KUKA KRL program: MyProgram_131().src

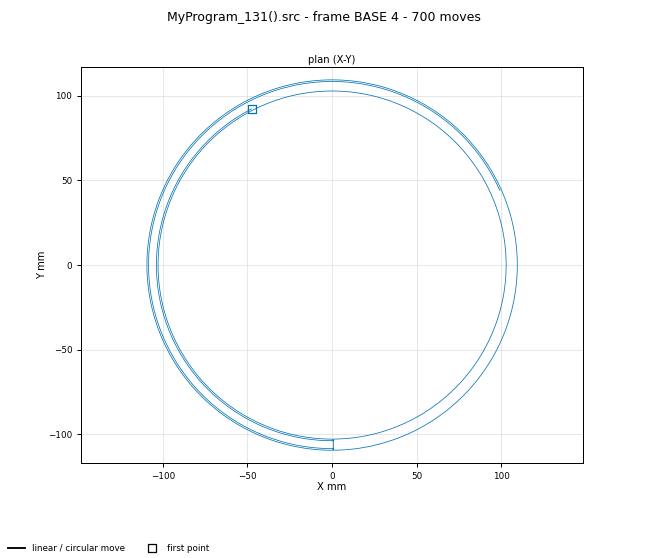
[picture p0: tool path of MyProgram_131().src in frame BASE 4, 700 of 700 moves have a stored position in this frame; points joined in program order, loops and branches not executed]
&ACCESS RVP
&REL 1
&PARAM TEMPLATE = C:\KRC\Roboter\Template\vorgabe
&PARAM EDITMASK = *
DEF MyProgram_131()
; ---- Setting reference (Base) ----
$BASE = BASE_DATA[4]

; --------------------------
; ---- Setting tool (TCP) ----
$TOOL = TOOL_DATA[3]
; --------------------------

$VEL.CP = VEL_APROX_PRINT
Startdeposition()
$VEL.CP = VEL_PRINT
LIN {X -47.5372,Y 92.2572,Z 107,A 112.7806,B 24.923,C -2.027,E1 24.926,E2 332.7039} C_DIS
LIN {X -49.4376,Y 91.2522,Z 107,A 114.1175,B 24.9227,C -2.0305,E1 24.9227,E2 331.3549} C_DIS
LIN {X -54.474,Y 88.3398,Z 107,A 117.7592,B 24.9219,C -2.0405,E1 24.9139,E2 327.6784} C_DIS
LIN {X -57.2487,Y 86.5659,Z 107,A 119.0499,B 24.9237,C -2.0176,E1 24.911,E2 326.4379} C_DIS
LIN {X -60.0172,Y 84.6705,Z 107,A 121.0764,B 24.9235,C -2.0203,E1 24.9063,E2 324.3982} C_DIS
LIN {X -63.2144,Y 82.3105,Z 107,A 123.2686,B 24.9238,C -2.0156,E1 24.9014,E2 322.2093} C_DIS
LIN {X -66.0188,Y 80.0795,Z 107,A 125.2015,B 24.9243,C -2.0096,E1 24.8973,E2 320.2834} C_DIS
LIN {X -68.7354,Y 77.7617,Z 107,A 127.217,B 24.9245,C -2.0067,E1 24.893,E2 318.2668} C_DIS
LIN {X -70.7621,Y 75.9209,Z 107,A 128.5161,B 24.9253,C -1.9956,E1 24.8904,E2 316.9891} C_DIS
LIN {X -72.935,Y 73.8345,Z 107,A 130.3237,B 24.9253,C -1.9968,E1 24.8867,E2 315.171} C_DIS
LIN {X -75.0796,Y 71.6545,Z 107,A 132.1843,B 24.9251,C -1.9988,E1 24.8831,E2 313.2975} C_DIS
LIN {X -77.6382,Y 68.8736,Z 107,A 134.0763,B 24.926,C -1.9866,E1 24.8796,E2 311.4263} C_DIS
LIN {X -79.2084,Y 67.061,Z 107,A 135.593,B 24.9257,C -1.9901,E1 24.8768,E2 309.8943} C_DIS
LIN {X -81.5466,Y 64.1968,Z 107,A 137.5851,B 24.9263,C -1.9829,E1 24.8734,E2 307.91} C_DIS
LIN {X -83.4567,Y 61.6949,Z 107,A 139.3497,B 24.9266,C -1.9792,E1 24.8704,E2 306.1458} C_DIS
LIN {X -85.5785,Y 58.7177,Z 107,A 141.2336,B 24.9273,C -1.9688,E1 24.8674,E2 304.2774} C_DIS
LIN {X -87.4411,Y 55.903,Z 107,A 143.96,B 24.9254,C -1.9945,E1 24.8632,E2 301.4758} C_DIS
LIN {X -89.8473,Y 51.948,Z 107,A 145.8018,B 24.9279,C -1.9615,E1 24.8607,E2 299.7033} C_DIS
LIN {X -91.4843,Y 49.0098,Z 107,A 148.2104,B 24.9268,C -1.9758,E1 24.8574,E2 297.2478} C_DIS
LIN {X -93.2578,Y 45.5457,Z 107,A 149.9432,B 24.9284,C -1.9545,E1 24.8554,E2 295.5565} C_DIS
LIN {X -94.9695,Y 41.8571,Z 107,A 151.8784,B 24.9297,C -1.9367,E1 24.8531,E2 293.6531} C_DIS
LIN {X -96.1628,Y 39.0355,Z 107,A 153.7151,B 24.9297,C -1.9367,E1 24.8512,E2 291.8063} C_DIS
LIN {X -97.0153,Y 36.8659,Z 107,A 155.0952,B 24.9297,C -1.936,E1 24.8498,E2 290.42} C_DIS
LIN {X -98.5087,Y 32.6703,Z 107,A 157.459,B 24.9305,C -1.925,E1 24.8476,E2 288.0691} C_DIS
LIN {X -99.5427,Y 29.3653,Z 107,A 159.4752,B 24.9307,C -1.9227,E1 24.846,E2 286.0467} C_DIS
LIN {X -100.6094,Y 25.4744,Z 107,A 161.5957,B 24.9315,C -1.9118,E1 24.8445,E2 283.9398} C_DIS
LIN {X -101.6647,Y 20.8647,Z 107,A 164.1136,B 24.9323,C -1.9002,E1 24.843,E2 281.4348} C_DIS
LIN {X -102.1521,Y 18.3302,Z 107,A 165.7626,B 24.9321,C -1.9035,E1 24.8421,E2 279.7681} C_DIS
LIN {X -102.734,Y 14.7241,Z 107,A 167.7191,B 24.9327,C -1.8949,E1 24.8413,E2 277.8206} C_DIS
LIN {X -103.1383,Y 11.5673,Z 107,A 169.4687,B 24.9331,C -1.889,E1 24.8407,E2 276.0746} C_DIS
LIN {X -103.3969,Y 8.9692,Z 107,A 171.1174,B 24.9329,C -1.8916,E1 24.8403,E2 274.4097} C_DIS
LIN {X -103.663,Y 5.0357,Z 107,A 173.3276,B 24.9333,C -1.8858,E1 24.8399,E2 272.2002} C_DIS
LIN {X -103.7792,Y 1.0625,Z 107,A 175.5136,B 24.9339,C -1.8784,E1 24.8398,E2 270.0186} C_DIS
LIN {X -103.7423,Y -2.9396,Z 107,A 177.7377,B 24.9343,C -1.8718,E1 24.8399,E2 267.7969} C_DIS
LIN {X -103.598,Y -6.2259,Z 107,A 179.5759,B 24.9347,C -1.8667,E1 24.8402,E2 265.9596} C_DIS
LIN {X -103.343,Y -9.5537,Z 107,A -178.6602,B 24.9353,C -1.8581,E1 24.8406,E2 264.2059} C_DIS
LIN {X -103.0312,Y -12.4821,Z 107,A -176.9436,B 24.9354,C -1.8561,E1 24.8412,E2 262.4836} C_DIS
LIN {X -102.5449,Y -15.9876,Z 107,A -175.0994,B 24.9361,C -1.8461,E1 24.8419,E2 260.6525} C_DIS
LIN {X -101.9172,Y -19.5943,Z 107,A -173.0077,B 24.9364,C -1.8422,E1 24.8429,E2 258.5575} C_DIS
LIN {X -101.3208,Y -22.4785,Z 107,A -171.4793,B 24.937,C -1.8337,E1 24.8438,E2 257.0404} C_DIS
LIN {X -100.5441,Y -25.7282,Z 107,A -169.5554,B 24.9372,C -1.8308,E1 24.8451,E2 255.1121} C_DIS
LIN {X -99.4164,Y -29.7911,Z 107,A -167.0771,B 24.9372,C -1.8291,E1 24.847,E2 252.6236} C_DIS
LIN {X -98.176,Y -33.6571,Z 107,A -164.8048,B 24.9377,C -1.8235,E1 24.849,E2 250.3518} C_DIS
LIN {X -96.8184,Y -37.3847,Z 107,A -162.589,B 24.9381,C -1.8179,E1 24.8512,E2 248.1366} C_DIS
LIN {X -95.3011,Y -41.0964,Z 107,A -160.5252,B 24.9389,C -1.8062,E1 24.8534,E2 246.0895} C_DIS
LIN {X -94.0744,Y -43.83,Z 107,A -158.8309,B 24.9391,C -1.8029,E1 24.8554,E2 244.3936} C_DIS
LIN {X -92.7841,Y -46.5012,Z 107,A -157.1505,B 24.9393,C -1.7999,E1 24.8575,E2 242.7115} C_DIS
LIN {X -90.1144,Y -51.4831,Z 107,A -154.2992,B 24.9405,C -1.7816,E1 24.8613,E2 239.8886} C_DIS
LIN {X -88.6267,Y -54.0034,Z 107,A -152.3658,B 24.94,C -1.7888,E1 24.8641,E2 237.9281} C_DIS
LIN {X -86.5659,Y -57.2487,Z 107,A -150.3857,B 24.9407,C -1.7781,E1 24.867,E2 235.9634} C_DIS
LIN {X -84.9538,Y -59.6164,Z 107,A -148.7985,B 24.941,C -1.7743,E1 24.8696,E2 234.3775} C_DIS
LIN {X -83.2306,Y -61.9991,Z 107,A -147.2699,B 24.9415,C -1.7669,E1 24.8721,E2 232.8592} C_DIS
LIN {X -81.4412,Y -64.3303,Z 107,A -145.4019,B 24.9412,C -1.7719,E1 24.8753,E2 230.9704} C_DIS
LIN {X -78.951,Y -67.3631,Z 107,A -143.2259,B 24.9415,C -1.7672,E1 24.8792,E2 228.7956} C_DIS
LIN {X -75.7408,Y -70.9536,Z 107,A -140.5603,B 24.9418,C -1.7615,E1 24.8842,E2 226.1318} C_DIS
LIN {X -73.0815,Y -73.6898,Z 107,A -138.0497,B 24.9412,C -1.7719,E1 24.8892,E2 223.5857} C_DIS
LIN {X -70.6358,Y -76.0396,Z 107,A -136.6878,B 24.9427,C -1.7492,E1 24.8919,E2 222.2724} C_DIS
LIN {X -68.8518,Y -77.6578,Z 107,A -135.1448,B 24.9423,C -1.7544,E1 24.8952,E2 220.7107} C_DIS
LIN {X -65.9356,Y -80.1487,Z 107,A -133.0147,B 24.9425,C -1.7509,E1 24.8997,E2 218.5809} C_DIS
LIN {X -63.4404,Y -82.1364,Z 107,A -131.372,B 24.943,C -1.7433,E1 24.9033,E2 216.9502} C_DIS
LIN {X -61.1951,Y -83.8226,Z 107,A -129.7963,B 24.9432,C -1.7416,E1 24.9068,E2 215.3731} C_DIS
LIN {X -58.2223,Y -85.914,Z 107,A -127.7657,B 24.9433,C -1.7391,E1 24.9115,E2 213.3413} C_DIS
LIN {X -55.7846,Y -87.5171,Z 107,A -126.1028,B 24.9433,C -1.7386,E1 24.9154,E2 211.6744} C_DIS
LIN {X -53.0914,Y -89.1766,Z 107,A -124.4049,B 24.9436,C -1.7342,E1 24.9195,E2 209.9818} C_DIS
LIN {X -49.2389,Y -91.36,Z 107,A -122.0744,B 24.9441,C -1.7265,E1 24.9251,E2 207.6627} C_DIS
LIN {X -46.3808,Y -92.8438,Z 107,A -120.1017,B 24.9438,C -1.7316,E1 24.9301,E2 205.6725} C_DIS
LIN {X -43.7788,Y -94.0982,Z 107,A -118.5776,B 24.9441,C -1.7271,E1 24.9339,E2 204.1554} C_DIS
LIN {X -40.3364,Y -95.6244,Z 107,A -116.4884,B 24.9442,C -1.7253,E1 24.9393,E2 202.0656} C_DIS
LIN {X -36.9737,Y -96.9745,Z 107,A -113.8939,B 24.9429,C -1.7461,E1 24.9462,E2 199.416} C_DIS
LIN {X -33.1975,Y -98.3309,Z 107,A -112.3467,B 24.9446,C -1.7186,E1 24.9501,E2 197.9313} C_DIS
LIN {X -30.1841,Y -99.299,Z 107,A -110.4082,B 24.9443,C -1.7246,E1 24.9553,E2 195.9751} C_DIS
LIN {X -26.4931,Y -100.347,Z 107,A -108.4997,B 24.9449,C -1.7152,E1 24.9604,E2 194.0861} C_DIS
LIN {X -23.4588,Y -101.0977,Z 107,A -106.603,B 24.9445,C -1.7209,E1 24.9656,E2 192.1732} C_DIS
LIN {X -19.4848,Y -101.9383,Z 107,A -104.3957,B 24.9446,C -1.7186,E1 24.9716,E2 189.9688} C_DIS
LIN {X -16.5691,Y -102.454,Z 107,A -102.6676,B 24.9444,C -1.7217,E1 24.9764,E2 188.2317} C_DIS
LIN {X -12.6661,Y -103.0096,Z 107,A -100.4703,B 24.9444,C -1.7221,E1 24.9825,E2 186.0318} C_DIS
LIN {X -8.6432,Y -103.4238,Z 107,A -98.2815,B 24.9445,C -1.7203,E1 24.9886,E2 183.8463} C_DIS
LIN {X -5.0186,Y -103.6638,Z 107,A -96.2028,B 24.9443,C -1.7232,E1 24.9944,E2 181.76} C_DIS
LIN {X -1.2387,Y -103.778,Z 107,A -94.3648,B 24.945,C -1.7137,E1 24.9995,E2 179.9443} C_DIS
LIN {X 0.7183,Y -103.7767,Z 107,A -93.2927,B 24.945,C -1.7137,E1 25.0025,E2 178.8722} C_DIS
Enddeposition()
LIN {X 0.7183,Y -103.7767,Z 107,A -93.2927,B 24.945,C -1.7137,E1 25.0025,E2 178.8722} C_DIS
Startdeposition()
$VEL.CP = VEL_PRINT
LIN {X -0.0761,Y -102.8201,Z 107,A -94.3958,B 24.9455,C -1.7047,E1 24.9993,E2 179.9968} C_DIS
LIN {X -2.5322,Y -102.7893,Z 107,A -95.9772,B 24.9461,C -1.6963,E1 24.9948,E2 181.5982} C_DIS
LIN {X -6.5744,Y -102.6089,Z 107,A -97.9527,B 24.9454,C -1.7068,E1 24.9894,E2 183.5492} C_DIS
LIN {X -8.8274,Y -102.4409,Z 107,A -99.4199,B 24.9459,C -1.6989,E1 24.9853,E2 185.0359} C_DIS
LIN {X -11.4014,Y -102.1861,Z 107,A -100.9306,B 24.9461,C -1.6964,E1 24.9811,E2 186.5534} C_DIS
LIN {X -15.1469,Y -101.6984,Z 107,A -102.8262,B 24.9455,C -1.7048,E1 24.9759,E2 188.4305} C_DIS
LIN {X -17.6331,Y -101.297,Z 107,A -104.2774,B 24.9456,C -1.7034,E1 24.9718,E2 189.8864} C_DIS
LIN {X -20.1263,Y -100.8311,Z 107,A -105.6747,B 24.9456,C -1.7046,E1 24.968,E2 191.2825} C_DIS
LIN {X -22.981,Y -100.2176,Z 107,A -107.1134,B 24.945,C -1.7125,E1 24.9641,E2 192.7043} C_DIS
LIN {X -25.0414,Y -99.7242,Z 107,A -108.4562,B 24.9454,C -1.707,E1 24.9605,E2 194.062} C_DIS
LIN {X -27.4771,Y -99.0808,Z 107,A -109.8639,B 24.9454,C -1.7077,E1 24.9567,E2 195.4701} C_DIS
LIN {X -30.3817,Y -98.2274,Z 107,A -111.6646,B 24.9455,C -1.7047,E1 24.9518,E2 197.2811} C_DIS
LIN {X -33.4794,Y -97.2171,Z 107,A -113.4221,B 24.9453,C -1.7083,E1 24.9472,E2 199.0332} C_DIS
LIN {X -35.8853,Y -96.3548,Z 107,A -114.8015,B 24.9451,C -1.7112,E1 24.9436,E2 200.4084} C_DIS
LIN {X -38.2411,Y -95.4443,Z 107,A -116.2076,B 24.9451,C -1.7126,E1 24.9399,E2 201.8143} C_DIS
LIN {X -40.566,Y -94.4796,Z 107,A -117.6131,B 24.9449,C -1.714,E1 24.9363,E2 203.2197} C_DIS
LIN {X -42.8147,Y -93.4824,Z 107,A -119.0182,B 24.9449,C -1.7142,E1 24.9327,E2 204.6277} C_DIS
LIN {X -45.158,Y -92.3729,Z 107,A -120.4656,B 24.9449,C -1.7159,E1 24.9291,E2 206.0749} C_DIS
LIN {X -47.3577,Y -91.265,Z 107,A -121.9236,B 24.9449,C -1.7144,E1 24.9254,E2 207.5402} C_DIS
LIN {X -49.6955,Y -90.0126,Z 107,A -123.2777,B 24.9445,C -1.721,E1 24.9221,E2 208.8826} C_DIS
LIN {X -51.8837,Y -88.7694,Z 107,A -124.6718,B 24.9443,C -1.7233,E1 24.9188,E2 210.2754} C_DIS
LIN {X -53.9437,Y -87.5337,Z 107,A -126.2088,B 24.9447,C -1.718,E1 24.9151,E2 211.8297} C_DIS
LIN {X -56.1184,Y -86.1552,Z 107,A -127.4851,B 24.9442,C -1.726,E1 24.9121,E2 213.0911} C_DIS
LIN {X -58.2109,Y -84.7555,Z 107,A -128.8962,B 24.944,C -1.728,E1 24.9088,E2 214.5022} C_DIS
LIN {X -60.2359,Y -83.3289,Z 107,A -130.3077,B 24.944,C -1.7292,E1 24.9056,E2 215.9157} C_DIS
LIN {X -62.724,Y -81.4701,Z 107,A -132.0601,B 24.9438,C -1.7315,E1 24.9017,E2 217.669} C_DIS
LIN {X -64.7681,Y -79.8546,Z 107,A -133.6037,B 24.9438,C -1.7308,E1 24.8983,E2 219.2199} C_DIS
LIN {X -67.1843,Y -77.835,Z 107,A -135.3788,B 24.9437,C -1.7334,E1 24.8946,E2 220.9956} C_DIS
LIN {X -69.5343,Y -75.7407,Z 107,A -137.0324,B 24.9432,C -1.7406,E1 24.8911,E2 222.6389} C_DIS
LIN {X -71.8178,Y -73.5816,Z 107,A -138.9911,B 24.9435,C -1.7368,E1 24.8872,E2 224.6148} C_DIS
LIN {X -74.1781,Y -71.1992,Z 107,A -140.7928,B 24.943,C -1.7432,E1 24.8837,E2 226.4089} C_DIS
LIN {X -76.611,Y -68.5743,Z 107,A -142.6677,B 24.9425,C -1.7519,E1 24.8802,E2 228.2713} C_DIS
LIN {X -78.2864,Y -66.6551,Z 107,A -144.1941,B 24.9425,C -1.7514,E1 24.8774,E2 229.8059} C_DIS
LIN {X -80.2918,Y -64.2283,Z 107,A -146.0563,B 24.9425,C -1.7517,E1 24.8741,E2 231.676} C_DIS
LIN {X -82.6132,Y -61.2134,Z 107,A -147.997,B 24.9417,C -1.7632,E1 24.8708,E2 233.5986} C_DIS
LIN {X -84.0655,Y -59.2035,Z 107,A -149.5834,B 24.942,C -1.7594,E1 24.8682,E2 235.2017} C_DIS
LIN {X -85.9185,Y -56.4775,Z 107,A -151.3261,B 24.9414,C -1.7675,E1 24.8656,E2 236.9339} C_DIS
LIN {X -87.5689,Y -53.8857,Z 107,A -152.9474,B 24.9409,C -1.7752,E1 24.8632,E2 238.5452} C_DIS
LIN {X -88.8623,Y -51.7252,Z 107,A -154.3501,B 24.9407,C -1.7789,E1 24.8612,E2 239.9462} C_DIS
LIN {X -90.0887,Y -49.5588,Z 107,A -155.7774,B 24.9405,C -1.7813,E1 24.8592,E2 241.3754} C_DIS
LIN {X -91.2661,Y -47.3557,Z 107,A -157.1569,B 24.9402,C -1.7855,E1 24.8574,E2 242.7521} C_DIS
LIN {X -92.4269,Y -45.0474,Z 107,A -158.7861,B 24.9404,C -1.7829,E1 24.8554,E2 244.3963} C_DIS
LIN {X -93.8431,Y -42.0144,Z 107,A -160.5575,B 24.9398,C -1.7915,E1 24.8534,E2 246.1569} C_DIS
LIN {X -94.9956,Y -39.3433,Z 107,A -162.1397,B 24.9394,C -1.7976,E1 24.8516,E2 247.7335} C_DIS
LIN {X -95.9307,Y -37.0049,Z 107,A -163.5255,B 24.9391,C -1.8023,E1 24.8502,E2 249.1158} C_DIS
LIN {X -96.8333,Y -34.573,Z 107,A -164.9482,B 24.9388,C -1.8073,E1 24.8489,E2 250.5345} C_DIS
LIN {X -97.6884,Y -32.0756,Z 107,A -166.3649,B 24.9383,C -1.8136,E1 24.8476,E2 251.9443} C_DIS
LIN {X -98.4067,Y -29.8015,Z 107,A -167.7742,B 24.9383,C -1.8148,E1 24.8464,E2 253.3588} C_DIS
LIN {X -99.1052,Y -27.3894,Z 107,A -169.257,B 24.9382,C -1.8162,E1 24.8453,E2 254.8469} C_DIS
LIN {X -99.7408,Y -24.9767,Z 107,A -170.6348,B 24.9378,C -1.8209,E1 24.8444,E2 256.2215} C_DIS
LIN {X -100.3228,Y -22.5256,Z 107,A -172.0196,B 24.9375,C -1.8259,E1 24.8435,E2 257.6025} C_DIS
LIN {X -100.8554,Y -20.0046,Z 107,A -173.4376,B 24.9372,C -1.831,E1 24.8427,E2 259.0167} C_DIS
LIN {X -101.3154,Y -17.5268,Z 107,A -175.0708,B 24.9374,C -1.8275,E1 24.8419,E2 260.6679} C_DIS
LIN {X -101.8931,Y -13.7765,Z 107,A -176.9788,B 24.9364,C -1.8413,E1 24.8411,E2 262.5544} C_DIS
LIN {X -102.2,Y -11.276,Z 107,A -178.4221,B 24.9362,C -1.8444,E1 24.8407,E2 263.9989} C_DIS
LIN {X -102.441,Y -8.826,Z 107,A -179.8044,B 24.936,C -1.8484,E1 24.8403,E2 265.3799} C_DIS
LIN {X -102.6593,Y -5.722,Z 107,A 178.6127,B 24.9352,C -1.8593,E1 24.84,E2 266.9466} C_DIS
LIN {X -102.7529,Y -3.7192,Z 107,A 177.3254,B 24.9354,C -1.8569,E1 24.8399,E2 268.2471} C_DIS
LIN {X -102.8138,Y -1.1098,Z 107,A 175.9089,B 24.9349,C -1.8629,E1 24.8398,E2 269.6578} C_DIS
LIN {X -102.811,Y 1.3581,Z 107,A 174.524,B 24.9347,C -1.867,E1 24.8398,E2 271.0413} C_DIS
LIN {X -102.7487,Y 3.8348,Z 107,A 173.0516,B 24.9346,C -1.8683,E1 24.8399,E2 272.5195} C_DIS
LIN {X -102.6227,Y 6.3692,Z 107,A 171.6611,B 24.9342,C -1.8737,E1 24.8402,E2 273.9055} C_DIS
LIN {X -102.3252,Y 10.0809,Z 107,A 169.5429,B 24.9338,C -1.8789,E1 24.8407,E2 276.024} C_DIS
LIN {X -102.0475,Y 12.5851,Z 107,A 168.1561,B 24.9335,C -1.8841,E1 24.8411,E2 277.4069} C_DIS
LIN {X -101.6997,Y 15.1383,Z 107,A 166.7368,B 24.9331,C -1.8893,E1 24.8417,E2 278.8222} C_DIS
LIN {X -101.2071,Y 18.133,Z 107,A 164.9234,B 24.933,C -1.8905,E1 24.8425,E2 280.6434} C_DIS
LIN {X -100.5717,Y 21.3843,Z 107,A 163.1798,B 24.9323,C -1.8999,E1 24.8435,E2 282.3748} C_DIS
LIN {X -100.0195,Y 23.8343,Z 107,A 161.7411,B 24.9321,C -1.903,E1 24.8444,E2 283.8146} C_DIS
LIN {X -99.4221,Y 26.2164,Z 107,A 160.3347,B 24.9319,C -1.9061,E1 24.8454,E2 285.2219} C_DIS
LIN {X -98.6158,Y 29.0968,Z 107,A 158.8866,B 24.931,C -1.9189,E1 24.8465,E2 286.6477} C_DIS
LIN {X -98.0043,Y 31.0994,Z 107,A 157.5095,B 24.9312,C -1.9153,E1 24.8476,E2 288.0414} C_DIS
LIN {X -97.2249,Y 33.4571,Z 107,A 156.0898,B 24.931,C -1.9184,E1 24.8489,E2 289.4619} C_DIS
LIN {X -96.3582,Y 35.8761,Z 107,A 154.6667,B 24.9307,C -1.9231,E1 24.8502,E2 290.8817} C_DIS
LIN {X -95.4461,Y 38.2365,Z 107,A 153.2833,B 24.9303,C -1.9284,E1 24.8516,E2 292.2603} C_DIS
LIN {X -94.4808,Y 40.5632,Z 107,A 151.8691,B 24.93,C -1.9323,E1 24.8532,E2 293.673} C_DIS
LIN {X -93.483,Y 42.8135,Z 107,A 150.4306,B 24.9299,C -1.9341,E1 24.8548,E2 295.115} C_DIS
LIN {X -92.3594,Y 45.1851,Z 107,A 148.8658,B 24.9299,C -1.935,E1 24.8567,E2 296.6863} C_DIS
LIN {X -91.2582,Y 47.3707,Z 107,A 147.5902,B 24.9293,C -1.9421,E1 24.8583,E2 297.9518} C_DIS
LIN {X -89.9448,Y 49.817,Z 107,A 145.9803,B 24.9291,C -1.9444,E1 24.8605,E2 299.5646} C_DIS
LIN {X -88.203,Y 52.842,Z 107,A 144.0992,B 24.9285,C -1.9523,E1 24.8631,E2 301.4367} C_DIS
LIN {X -86.866,Y 55.0124,Z 107,A 142.6426,B 24.9283,C -1.955,E1 24.8653,E2 302.8942} C_DIS
LIN {X -85.4922,Y 57.124,Z 107,A 141.2293,B 24.9281,C -1.9586,E1 24.8675,E2 304.306} C_DIS
LIN {X -83.7242,Y 59.6819,Z 107,A 139.4889,B 24.9277,C -1.9632,E1 24.8702,E2 306.0441} C_DIS
LIN {X -81.8245,Y 62.2641,Z 107,A 137.5093,B 24.9279,C -1.9613,E1 24.8736,E2 308.0378} C_DIS
LIN {X -79.8595,Y 64.7621,Z 107,A 135.8362,B 24.9273,C -1.9694,E1 24.8765,E2 309.6993} C_DIS
LIN {X -77.5417,Y 67.5202,Z 107,A 133.8707,B 24.9268,C -1.976,E1 24.88,E2 311.6579} C_DIS
LIN {X -75.7336,Y 69.5421,Z 107,A 132.296,B 24.9267,C -1.9777,E1 24.883,E2 313.2358} C_DIS
LIN {X -73.5691,Y 71.8305,Z 107,A 130.435,B 24.9267,C -1.9782,E1 24.8866,E2 315.1034} C_DIS
LIN {X -71.334,Y 74.0482,Z 107,A 128.7682,B 24.9261,C -1.9856,E1 24.8899,E2 316.7598} C_DIS
LIN {X -69.0197,Y 76.2122,Z 107,A 127.0945,B 24.9255,C -1.9929,E1 24.8933,E2 318.4228} C_DIS
LIN {X -66.6975,Y 78.2503,Z 107,A 125.3489,B 24.9253,C -1.996,E1 24.897,E2 320.168} C_DIS
LIN {X -64.2483,Y 80.2759,Z 107,A 123.3745,B 24.9256,C -1.9926,E1 24.9013,E2 322.1577} C_DIS
LIN {X -61.2094,Y 82.6161,Z 107,A 121.4285,B 24.9247,C -2.0039,E1 24.9056,E2 324.0838} C_DIS
LIN {X -59.1996,Y 84.0682,Z 107,A 119.8927,B 24.9249,C -2.0012,E1 24.9091,E2 325.6313} C_DIS
LIN {X -57.1201,Y 85.4948,Z 107,A 118.4125,B 24.9249,C -2.0013,E1 24.9126,E2 327.1163} C_DIS
LIN {X -54.6975,Y 87.0628,Z 107,A 117.07,B 24.924,C -2.0139,E1 24.9157,E2 328.4332} C_DIS
LIN {X -52.7036,Y 88.2848,Z 107,A 115.7335,B 24.9239,C -2.015,E1 24.9189,E2 329.771} C_DIS
LIN {X -50.173,Y 89.746,Z 107,A 113.9977,B 24.9239,C -2.0141,E1 24.9231,E2 331.5142} C_DIS
LIN {X -47.3316,Y 91.2785,Z 107,A 112.2752,B 24.9235,C -2.0198,E1 24.9273,E2 333.2278} C_DIS
LIN {X -45.0322,Y 92.4342,Z 107,A 110.836,B 24.9233,C -2.022,E1 24.9309,E2 334.6658} C_DIS
LIN {X -42.7562,Y 93.5088,Z 107,A 109.4575,B 24.9231,C -2.025,E1 24.9344,E2 336.0405} C_DIS
LIN {X -40.4541,Y 94.5275,Z 107,A 108.0504,B 24.923,C -2.0269,E1 24.938,E2 337.4464} C_DIS
LIN {X -38.1031,Y 95.4994,Z 107,A 106.6306,B 24.9228,C -2.0288,E1 24.9417,E2 338.8648} C_DIS
LIN {X -35.8145,Y 96.3814,Z 107,A 105.1647,B 24.923,C -2.027,E1 24.9455,E2 340.338} C_DIS
LIN {X -33.3842,Y 97.2496,Z 107,A 103.7931,B 24.9226,C -2.0312,E1 24.9491,E2 341.7023} C_DIS
LIN {X -31.0175,Y 98.0303,Z 107,A 102.371,B 24.9226,C -2.0316,E1 24.9529,E2 343.1259} C_DIS
LIN {X -28.6258,Y 98.7553,Z 107,A 100.9714,B 24.9226,C -2.0329,E1 24.9566,E2 344.5248} C_DIS
LIN {X -26.2156,Y 99.4223,Z 107,A 99.4611,B 24.9227,C -2.0301,E1 24.9607,E2 346.0442} C_DIS
LIN {X -23.6931,Y 100.0531,Z 107,A 98.1781,B 24.9222,C -2.0375,E1 24.9642,E2 347.3112} C_DIS
LIN {X -21.2911,Y 100.592,Z 107,A 96.7464,B 24.9222,C -2.0365,E1 24.9681,E2 348.7471} C_DIS
LIN {X -18.8187,Y 101.0837,Z 107,A 95.194,B 24.9226,C -2.0322,E1 24.9724,E2 350.3114} C_DIS
LIN {X -16.3161,Y 101.5176,Z 107,A 93.9222,B 24.9221,C -2.0385,E1 24.9759,E2 351.5695} C_DIS
LIN {X -13.769,Y 101.8941,Z 107,A 92.5423,B 24.9218,C -2.0415,E1 24.9797,E2 352.9434} C_DIS
LIN {X -11.2698,Y 102.2007,Z 107,A 91.108,B 24.9218,C -2.0411,E1 24.9836,E2 354.3795} C_DIS
LIN {X -8.8208,Y 102.4415,Z 107,A 89.7197,B 24.9218,C -2.0411,E1 24.9875,E2 355.7685} C_DIS
LIN {X -6.2228,Y 102.6316,Z 107,A 88.3123,B 24.9218,C -2.0434,E1 24.9914,E2 357.171} C_DIS
LIN {X -3.7107,Y 102.7532,Z 107,A 86.8805,B 24.9218,C -2.0428,E1 24.9954,E2 358.6047} C_DIS
LIN {X -1.2528,Y 102.8129,Z 107,A 85.4815,B 24.9218,C -2.042,E1 24.9993,E2 360.0056} C_DIS
LIN {X 1.2636,Y 102.8128,Z 107,A 84.1059,B 24.9218,C -2.0433,E1 25.0032,E2 361.3781} C_DIS
LIN {X 4.1048,Y 102.7371,Z 107,A 82.6802,B 24.9212,C -2.0494,E1 25.0071,E2 362.789} C_DIS
LIN {X 6.366,Y 102.6229,Z 107,A 81.2553,B 24.9217,C -2.0432,E1 25.0111,E2 364.228} C_DIS
LIN {X 8.831,Y 102.4406,Z 107,A 79.8831,B 24.9217,C -2.0433,E1 25.0149,E2 365.5992} C_DIS
LIN {X 11.3946,Y 102.1869,Z 107,A 78.4773,B 24.9217,C -2.0443,E1 25.0188,E2 367.0018} C_DIS
LIN {X 13.8376,Y 101.8852,Z 107,A 77.0488,B 24.9218,C -2.0418,E1 25.0228,E2 368.4351} C_DIS
LIN {X 16.3452,Y 101.513,Z 107,A 75.637,B 24.9218,C -2.0414,E1 25.0267,E2 369.8464} C_DIS
LIN {X 20.1218,Y 100.8321,Z 107,A 73.5282,B 24.9218,C -2.0417,E1 25.0325,E2 371.9522} C_DIS
LIN {X 22.5302,Y 100.3218,Z 107,A 72.1298,B 24.922,C -2.04,E1 25.0363,E2 373.3527} C_DIS
LIN {X 25.0369,Y 99.7254,Z 107,A 70.7511,B 24.9219,C -2.0413,E1 25.04,E2 374.7262} C_DIS
LIN {X 27.9988,Y 98.933,Z 107,A 69.0753,B 24.9219,C -2.0415,E1 25.0445,E2 376.399} C_DIS
LIN {X 32.3214,Y 97.6079,Z 107,A 66.4051,B 24.9224,C -2.0337,E1 25.0517,E2 379.0828} C_DIS
LIN {X 34.7048,Y 96.7862,Z 107,A 65.1007,B 24.9222,C -2.0363,E1 25.0551,E2 380.3783} C_DIS
LIN {X 37.4439,Y 95.7583,Z 107,A 63.668,B 24.9218,C -2.0425,E1 25.0588,E2 381.7934} C_DIS
LIN {X 39.3465,Y 94.9943,Z 107,A 62.3066,B 24.9225,C -2.0327,E1 25.0623,E2 383.1747} C_DIS
LIN {X 41.6755,Y 93.9958,Z 107,A 60.9249,B 24.9225,C -2.0323,E1 25.0659,E2 384.554} C_DIS
LIN {X 43.9657,Y 92.9466,Z 107,A 59.357,B 24.9232,C -2.0243,E1 25.0699,E2 386.137} C_DIS
LIN {X 46.2823,Y 91.8147,Z 107,A 58.1209,B 24.9227,C -2.0303,E1 25.0729,E2 387.3555} C_DIS
LIN {X 48.5186,Y 90.6529,Z 107,A 56.6832,B 24.9229,C -2.0271,E1 25.0765,E2 388.7967} C_DIS
LIN {X 50.6885,Y 89.458,Z 107,A 55.316,B 24.9231,C -2.0257,E1 25.0798,E2 390.1632} C_DIS
LIN {X 52.8623,Y 88.1909,Z 107,A 53.9178,B 24.9232,C -2.0238,E1 25.0832,E2 391.5617} C_DIS
LIN {X 55.0045,Y 86.871,Z 107,A 52.3195,B 24.9239,C -2.0139,E1 25.087,E2 393.1782} C_DIS
LIN {X 58.2198,Y 84.7493,Z 107,A 50.4097,B 24.9235,C -2.0197,E1 25.0914,E2 395.0678} C_DIS
LIN {X 61.2677,Y 82.5731,Z 107,A 48.289,B 24.9239,C -2.0148,E1 25.0962,E2 397.1928} C_DIS
LIN {X 63.7379,Y 80.6793,Z 107,A 46.5593,B 24.9241,C -2.0119,E1 25.1,E2 398.923} C_DIS
LIN {X 66.2039,Y 78.6708,Z 107,A 44.6334,B 24.9248,C -2.0023,E1 25.1042,E2 400.8641} C_DIS
LIN {X 68.6217,Y 76.5685,Z 107,A 42.9212,B 24.9248,C -2.0017,E1 25.1078,E2 402.5709} C_DIS
LIN {X 71.3614,Y 74.0218,Z 107,A 40.8606,B 24.9251,C -1.9984,E1 25.1119,E2 404.631} C_DIS
LIN {X 73.6272,Y 71.7708,Z 107,A 38.9931,B 24.9257,C -1.991,E1 25.1156,E2 406.5079} C_DIS
LIN {X 75.7641,Y 69.5088,Z 107,A 37.4052,B 24.9255,C -1.993,E1 25.1186,E2 408.0841} C_DIS
LIN {X 77.8562,Y 67.1601,Z 107,A 35.7018,B 24.9257,C -1.991,E1 25.1218,E2 409.7847} C_DIS
LIN {X 79.8546,Y 64.7682,Z 107,A 33.9675,B 24.926,C -1.987,E1 25.1249,E2 411.5204} C_DIS
LIN {X 81.8294,Y 62.2576,Z 107,A 32.1875,B 24.9263,C -1.9826,E1 25.1279,E2 413.3023} C_DIS
LIN {X 84.0786,Y 59.1846,Z 107,A 30.0793,B 24.9267,C -1.9779,E1 25.1313,E2 415.4115} C_DIS
LIN {X 85.4998,Y 57.1125,Z 107,A 28.6866,B 24.9269,C -1.9746,E1 25.1335,E2 416.805} C_DIS
LIN {X 86.9008,Y 54.9568,Z 107,A 27.1789,B 24.9274,C -1.9678,E1 25.1358,E2 418.3212} C_DIS
LIN {X 88.2184,Y 52.816,Z 107,A 25.7032,B 24.9279,C -1.961,E1 25.138,E2 419.8053} C_DIS
LIN {X 90.2064,Y 49.3417,Z 107,A 23.7767,B 24.9274,C -1.9674,E1 25.1406,E2 421.7069} C_DIS
LIN {X 91.2682,Y 47.3517,Z 107,A 22.3105,B 24.9283,C -1.9553,E1 25.1425,E2 423.1937} C_DIS
LIN {X 92.4394,Y 45.0215,Z 107,A 20.9857,B 24.9283,C -1.9565,E1 25.1441,E2 424.5087} C_DIS
LIN {X 93.5116,Y 42.75,Z 107,A 19.6231,B 24.9284,C -1.9541,E1 25.1457,E2 425.8697} C_DIS
LIN {X 94.5286,Y 40.4517,Z 107,A 18.2318,B 24.9287,C -1.9504,E1 25.1473,E2 427.2621} C_DIS
LIN {X 95.5068,Y 38.0841,Z 107,A 16.8332,B 24.9289,C -1.9474,E1 25.1488,E2 428.66} C_DIS
LIN {X 96.3729,Y 35.8373,Z 107,A 15.348,B 24.9296,C -1.9376,E1 25.1502,E2 430.1601} C_DIS
LIN {X 97.2286,Y 33.4466,Z 107,A 14.0434,B 24.9296,C -1.9379,E1 25.1514,E2 431.4567} C_DIS
LIN {X 98.0188,Y 31.0545,Z 107,A 12.4686,B 24.9304,C -1.9266,E1 25.1528,E2 433.0491} C_DIS
LIN {X 98.9734,Y 27.8563,Z 107,A 10.7358,B 24.9304,C -1.9262,E1 25.1541,E2 434.773} C_DIS
LIN {X 99.74,Y 24.98,Z 107,A 9.1254,B 24.9307,C -1.9231,E1 25.1553,E2 436.3815} C_DIS
LIN {X 100.3219,Y 22.5294,Z 107,A 7.7578,B 24.9309,C -1.9202,E1 25.1561,E2 437.7479} C_DIS
LIN {X 100.8593,Y 19.9844,Z 107,A 6.3487,B 24.9311,C -1.9173,E1 25.1569,E2 439.1556} C_DIS
LIN {X 101.3182,Y 17.5101,Z 107,A 4.9559,B 24.9314,C -1.9133,E1 25.1576,E2 440.5497} C_DIS
LIN {X 101.7602,Y 14.7171,Z 107,A 3.5096,B 24.9314,C -1.9137,E1 25.1582,E2 441.9865} C_DIS
LIN {X 102.0472,Y 12.5871,Z 107,A 2.1449,B 24.9321,C -1.903,E1 25.1587,E2 443.3686} C_DIS
LIN {X 102.3363,Y 9.9611,Z 107,A 0.7648,B 24.9321,C -1.9021,E1 25.1591,E2 444.7426} C_DIS
LIN {X 102.5421,Y 7.5616,Z 107,A -0.6635,B 24.9327,C -1.8942,E1 25.1594,E2 446.1811} C_DIS
LIN {X 102.6976,Y 5.0238,Z 107,A -2.0552,B 24.933,C -1.8907,E1 25.1596,E2 447.5727} C_DIS
LIN {X 102.7982,Y 2.0546,Z 107,A -3.5343,B 24.9328,C -1.8927,E1 25.1598,E2 449.0383} C_DIS
LIN {X 102.82,Y 0.0038,Z 107,A -4.8043,B 24.9335,C -1.8837,E1 25.1598,E2 450.322} C_DIS
LIN {X 102.7889,Y -2.5475,Z 107,A -6.2469,B 24.9339,C -1.8782,E1 25.1598,E2 451.7689} C_DIS
LIN {X 102.6959,Y -5.0603,Z 107,A -7.6388,B 24.9342,C -1.8741,E1 25.1595,E2 453.1623} C_DIS
LIN {X 102.5368,Y -7.6281,Z 107,A -9.1676,B 24.9348,C -1.8655,E1 25.1592,E2 454.7023} C_DIS
LIN {X 102.3255,Y -10.0775,Z 107,A -10.4227,B 24.9348,C -1.8658,E1 25.1589,E2 455.9492} C_DIS
LIN {X 102.0483,Y -12.5779,Z 107,A -11.795,B 24.935,C -1.8625,E1 25.1585,E2 457.3213} C_DIS
LIN {X 101.6975,Y -15.1525,Z 107,A -13.1969,B 24.9352,C -1.8597,E1 25.1579,E2 458.7214} C_DIS
LIN {X 101.2959,Y -17.6391,Z 107,A -14.7874,B 24.936,C -1.8474,E1 25.1572,E2 460.3315} C_DIS
LIN {X 100.8334,Y -20.1153,Z 107,A -16.0139,B 24.9358,C -1.8502,E1 25.1565,E2 461.5441} C_DIS
LIN {X 100.3233,Y -22.5234,Z 107,A -17.4016,B 24.9362,C -1.8452,E1 25.1557,E2 462.9357} C_DIS
LIN {X 99.7273,Y -25.0296,Z 107,A -18.7786,B 24.9363,C -1.843,E1 25.1548,E2 464.3099} C_DIS
LIN {X 98.9521,Y -27.9313,Z 107,A -20.5131,B 24.9369,C -1.8352,E1 25.1535,E2 466.0529} C_DIS
LIN {X 97.9991,Y -31.1155,Z 107,A -22.3206,B 24.9371,C -1.8312,E1 25.152,E2 467.8595} C_DIS
LIN {X 97.2198,Y -33.4716,Z 107,A -23.6966,B 24.9374,C -1.8271,E1 25.1508,E2 469.2373} C_DIS
LIN {X 96.3493,Y -35.8997,Z 107,A -25.0742,B 24.9376,C -1.8251,E1 25.1495,E2 470.612} C_DIS
LIN {X 95.4435,Y -38.243,Z 107,A -26.4651,B 24.9378,C -1.8212,E1 25.1481,E2 472.0045} C_DIS
LIN {X 94.4804,Y -40.5643,Z 107,A -27.8578,B 24.9381,C -1.8172,E1 25.1466,E2 473.3989} C_DIS
LIN {X 93.4848,Y -42.8094,Z 107,A -29.2472,B 24.9384,C -1.8122,E1 25.145,E2 474.7926} C_DIS
LIN {X 92.3858,Y -45.1318,Z 107,A -30.6817,B 24.9387,C -1.8077,E1 25.1432,E2 476.2299} C_DIS
LIN {X 91.2664,Y -47.3551,Z 107,A -32.0746,B 24.939,C -1.8033,E1 25.1414,E2 477.6257} C_DIS
LIN {X 90.0504,Y -49.6278,Z 107,A -33.637,B 24.9397,C -1.7939,E1 25.1393,E2 479.2021} C_DIS
LIN {X 88.3934,Y -52.5199,Z 107,A -35.3729,B 24.9397,C -1.7935,E1 25.1369,E2 480.93} C_DIS
LIN {X 86.8651,Y -55.0137,Z 107,A -36.9672,B 24.9399,C -1.7903,E1 25.1346,E2 482.5239} C_DIS
LIN {X 85.4918,Y -57.1246,Z 107,A -38.3621,B 24.9402,C -1.7867,E1 25.1324,E2 483.9204} C_DIS
LIN {X 84.0457,Y -59.2313,Z 107,A -39.748,B 24.9403,C -1.7843,E1 25.1302,E2 485.3051} C_DIS
LIN {X 82.5734,Y -61.2673,Z 107,A -41.1541,B 24.9406,C -1.7802,E1 25.1279,E2 486.7141} C_DIS
LIN {X 80.6798,Y -63.7372,Z 107,A -42.8804,B 24.9409,C -1.7759,E1 25.1249,E2 488.4425} C_DIS
LIN {X 78.6754,Y -66.1986,Z 107,A -44.6499,B 24.9412,C -1.7712,E1 25.1218,E2 490.2149} C_DIS
LIN {X 76.9796,Y -68.1625,Z 107,A -46.0595,B 24.9414,C -1.7689,E1 25.1192,E2 491.6235} C_DIS
LIN {X 74.8865,Y -70.4534,Z 107,A -47.8832,B 24.9419,C -1.7607,E1 25.1157,E2 493.4586} C_DIS
LIN {X 72.3503,Y -73.0556,Z 107,A -49.8414,B 24.942,C -1.7584,E1 25.1119,E2 495.4137} C_DIS
LIN {X 69.9854,Y -75.3266,Z 107,A -51.6444,B 24.9423,C -1.755,E1 25.1082,E2 497.2174} C_DIS
LIN {X 68.069,Y -77.0624,Z 107,A -53.238,B 24.9429,C -1.7455,E1 25.1048,E2 498.8272} C_DIS
LIN {X 65.6837,Y -79.1033,Z 107,A -54.8886,B 24.9429,C -1.7455,E1 25.1013,E2 500.4713} C_DIS
LIN {X 62.2153,Y -81.8612,Z 107,A -57.4134,B 24.9434,C -1.7379,E1 25.0958,E2 503.0048} C_DIS
LIN {X 60.1711,Y -83.3752,Z 107,A -58.628,B 24.9431,C -1.7431,E1 25.0931,E2 504.2027} C_DIS
LIN {X 58.112,Y -84.8232,Z 107,A -60.0246,B 24.9432,C -1.7405,E1 25.0899,E2 505.6007} C_DIS
LIN {X 56.0177,Y -86.2207,Z 107,A -61.4508,B 24.9435,C -1.7368,E1 25.0865,E2 507.0309} C_DIS
LIN {X 53.8896,Y -87.5666,Z 107,A -62.8481,B 24.9436,C -1.7344,E1 25.0832,E2 508.4296} C_DIS
LIN {X 51.7292,Y -88.86,Z 107,A -64.2208,B 24.9437,C -1.733,E1 25.0799,E2 509.8012} C_DIS
LIN {X 49.1505,Y -90.3101,Z 107,A -65.6906,B 24.9434,C -1.7373,E1 25.0764,E2 511.2566} C_DIS
LIN {X 47.348,Y -91.2701,Z 107,A -67.1955,B 24.9445,C -1.7206,E1 25.0726,E2 512.7968} C_DIS
LIN {X 45.0019,Y -92.4487,Z 107,A -68.4765,B 24.9442,C -1.7255,E1 25.0694,E2 514.0628} C_DIS
LIN {X 42.7355,Y -93.5181,Z 107,A -69.8409,B 24.9442,C -1.7246,E1 25.0659,E2 515.4258} C_DIS
LIN {X 40.4404,Y -94.5333,Z 107,A -71.2349,B 24.9444,C -1.7227,E1 25.0624,E2 516.821} C_DIS
LIN {X 38.1196,Y -95.4928,Z 107,A -72.6286,B 24.9445,C -1.7209,E1 25.0587,E2 518.2158} C_DIS
LIN {X 35.7072,Y -96.4205,Z 107,A -74.1048,B 24.9447,C -1.7175,E1 25.0549,E2 519.6967} C_DIS
LIN {X 33.3986,Y -97.2447,Z 107,A -75.4471,B 24.9447,C -1.7167,E1 25.0513,E2 521.0383} C_DIS
LIN {X 31.0505,Y -98.0201,Z 107,A -76.8501,B 24.9449,C -1.714,E1 25.0476,E2 522.445} C_DIS
LIN {X 28.6355,Y -98.7526,Z 107,A -78.2642,B 24.9451,C -1.7121,E1 25.0438,E2 523.8612} C_DIS
LIN {X 26.2057,Y -99.425,Z 107,A -79.8439,B 24.9456,C -1.7037,E1 25.0395,E2 525.4583} C_DIS
LIN {X 22.5151,Y -100.3251,Z 107,A -81.7502,B 24.9452,C -1.7099,E1 25.0344,E2 527.3472} C_DIS
LIN {X 19.9948,Y -100.8573,Z 107,A -83.1539,B 24.9452,C -1.7099,E1 25.0305,E2 528.7491} C_DIS
LIN {X 17.5183,Y -101.3169,Z 107,A -84.5547,B 24.9452,C -1.7089,E1 25.0267,E2 530.1508} C_DIS
LIN {X 14.9998,Y -101.7201,Z 107,A -86.002,B 24.9454,C -1.7069,E1 25.0227,E2 531.6015} C_DIS
LIN {X 12.5653,Y -102.0498,Z 107,A -87.3971,B 24.9455,C -1.7049,E1 25.0188,E2 533.0001} C_DIS
LIN {X 8.8125,Y -102.4422,Z 107,A -89.4697,B 24.9455,C -1.7049,E1 25.0131,E2 535.0713} C_DIS
LIN {X 6.2458,Y -102.6303,Z 107,A -90.939,B 24.9457,C -1.703,E1 25.009,E2 536.5447} C_DIS
LIN {X 3.6903,Y -102.7538,Z 107,A -92.3258,B 24.9456,C -1.7039,E1 25.0051,E2 537.9287} C_DIS
LIN {X 0.7131,Y -102.8158,Z 107,A -93.7448,B 24.945,C -1.7128,E1 25.0012,E2 539.3266} C_DIS
Enddeposition()
LIN {X 0.7596,Y -109.3904,Z 108,A -93.4503,B 24.951,C -1.6165,E1 25.0014,E2 539.2604} C_DIS
Startdeposition()
$VEL.CP = VEL_PRINT
LIN {X 2.6847,Y -109.3625,Z 108,A -92.0814,B 24.9501,C -1.6318,E1 25.0053,E2 537.8553} C_DIS
LIN {X 5.3678,Y -109.2636,Z 108,A -90.6764,B 24.9501,C -1.6323,E1 25.0092,E2 536.4497} C_DIS
LIN {X 8.0476,Y -109.099,Z 108,A -89.2933,B 24.9501,C -1.632,E1 25.0131,E2 535.068} C_DIS
LIN {X 11.1782,Y -108.8209,Z 108,A -87.8346,B 24.9505,C -1.625,E1 25.0171,E2 533.6267} C_DIS
LIN {X 13.3912,Y -108.5727,Z 108,A -86.39,B 24.9498,C -1.6374,E1 25.0212,E2 532.1537} C_DIS
LIN {X 16.0996,Y -108.204,Z 108,A -85.0782,B 24.95,C -1.6333,E1 25.0248,E2 530.8527} C_DIS
LIN {X 19.1759,Y -107.6997,Z 108,A -83.6197,B 24.9504,C -1.6272,E1 25.0287,E2 529.4103} C_DIS
LIN {X 21.3895,Y -107.2837,Z 108,A -82.2476,B 24.9498,C -1.6364,E1 25.0325,E2 528.0181} C_DIS
LIN {X 24.0159,Y -106.7264,Z 108,A -80.8439,B 24.9498,C -1.6375,E1 25.0364,E2 526.6135} C_DIS
LIN {X 26.6279,Y -106.1049,Z 108,A -79.4639,B 24.9498,C -1.6378,E1 25.0401,E2 525.2348} C_DIS
LIN {X 29.1772,Y -105.4327,Z 108,A -78.063,B 24.9496,C -1.6402,E1 25.0439,E2 523.8306} C_DIS
LIN {X 31.8021,Y -104.6705,Z 108,A -76.6351,B 24.9496,C -1.6416,E1 25.0477,E2 522.4016} C_DIS
LIN {X 34.3613,Y -103.8585,Z 108,A -75.2321,B 24.9494,C -1.6432,E1 25.0515,E2 520.9976} C_DIS
LIN {X 36.8542,Y -103.0006,Z 108,A -73.6653,B 24.9488,C -1.653,E1 25.0556,E2 519.4108} C_DIS
LIN {X 39.416,Y -102.0474,Z 108,A -72.451,B 24.9493,C -1.6456,E1 25.0588,E2 518.2166} C_DIS
LIN {X 41.8638,Y -101.0682,Z 108,A -71.0513,B 24.9491,C -1.6484,E1 25.0624,E2 516.8136} C_DIS
LIN {X 44.3315,Y -100.0104,Z 108,A -69.6273,B 24.9489,C -1.6513,E1 25.066,E2 515.3861} C_DIS
LIN {X 46.7726,Y -98.8923,Z 108,A -68.2481,B 24.9489,C -1.6523,E1 25.0695,E2 514.0079} C_DIS
LIN {X 49.1854,Y -97.7146,Z 108,A -66.8472,B 24.9487,C -1.6544,E1 25.073,E2 512.6059} C_DIS
LIN {X 51.6113,Y -96.455,Z 108,A -65.4439,B 24.9487,C -1.6557,E1 25.0765,E2 511.2036} C_DIS
LIN {X 53.9208,Y -95.1835,Z 108,A -64.0227,B 24.9484,C -1.6599,E1 25.08,E2 509.7766} C_DIS
LIN {X 56.2819,Y -93.8064,Z 108,A -62.5373,B 24.9481,C -1.6649,E1 25.0836,E2 508.284} C_DIS
LIN {X 58.5263,Y -92.4231,Z 108,A -61.2218,B 24.9481,C -1.6647,E1 25.0867,E2 506.9732} C_DIS
LIN {X 61.1743,Y -90.6898,Z 108,A -59.7871,B 24.9485,C -1.6582,E1 25.09,E2 505.5585} C_DIS
LIN {X 63.3294,Y -89.1985,Z 108,A -58.4239,B 24.9483,C -1.6606,E1 25.0931,E2 504.1943} C_DIS
LIN {X 65.1668,Y -87.8672,Z 108,A -57.0435,B 24.9476,C -1.6715,E1 25.0962,E2 502.7931} C_DIS
LIN {X 67.3035,Y -86.2415,Z 108,A -55.6216,B 24.9474,C -1.6752,E1 25.0994,E2 501.3676} C_DIS
LIN {X 69.3997,Y -84.5638,Z 108,A -54.2442,B 24.9473,C -1.6771,E1 25.1024,E2 499.991} C_DIS
LIN {X 71.8833,Y -82.4604,Z 108,A -52.7806,B 24.9477,C -1.6704,E1 25.1054,E2 498.5489} C_DIS
LIN {X 73.5012,Y -81.0239,Z 108,A -51.4436,B 24.947,C -1.682,E1 25.1083,E2 497.19} C_DIS
LIN {X 75.8331,Y -78.8432,Z 108,A -49.9839,B 24.9473,C -1.6766,E1 25.1112,E2 495.7488} C_DIS
LIN {X 77.3542,Y -77.3542,Z 108,A -48.648,B 24.9465,C -1.6891,E1 25.1139,E2 494.3892} C_DIS
LIN {X 79.2625,Y -75.3972,Z 108,A -47.2469,B 24.9464,C -1.6913,E1 25.1166,E2 492.9889} C_DIS
LIN {X 81.0567,Y -73.4655,Z 108,A -45.8282,B 24.9461,C -1.6965,E1 25.1193,E2 491.5642} C_DIS
LIN {X 82.8666,Y -71.4172,Z 108,A -44.427,B 24.9459,C -1.6989,E1 25.1219,E2 490.1637} C_DIS
LIN {X 84.5638,Y -69.3997,Z 108,A -43.0315,B 24.9456,C -1.7032,E1 25.1244,E2 488.7645} C_DIS
LIN {X 86.4544,Y -67.0272,Z 108,A -41.6098,B 24.9458,C -1.7,E1 25.1268,E2 487.3569} C_DIS
LIN {X 87.8959,Y -65.1276,Z 108,A -40.2326,B 24.9453,C -1.7091,E1 25.1291,E2 485.9648} C_DIS
LIN {X 89.44,Y -62.9908,Z 108,A -38.8375,B 24.945,C -1.7136,E1 25.1314,E2 484.566} C_DIS
LIN {X 90.959,Y -60.7768,Z 108,A -37.4398,B 24.9447,C -1.7171,E1 25.1336,E2 483.1668} C_DIS
LIN {X 92.4231,Y -58.5263,Z 108,A -36.0644,B 24.9446,C -1.7198,E1 25.1356,E2 481.7921} C_DIS
LIN {X 93.8316,Y -56.2405,Z 108,A -34.6445,B 24.9443,C -1.7245,E1 25.1377,E2 480.3684} C_DIS
LIN {X 95.2072,Y -53.8785,Z 108,A -33.2671,B 24.9442,C -1.7262,E1 25.1396,E2 478.9939} C_DIS
LIN {X 96.5007,Y -51.5257,Z 108,A -31.7185,B 24.9435,C -1.7368,E1 25.1417,E2 477.4286} C_DIS
LIN {X 97.7362,Y -49.142,Z 108,A -30.4497,B 24.9435,C -1.7348,E1 25.1433,E2 476.1711} C_DIS
LIN {X 98.8923,Y -46.7726,Z 108,A -29.0553,B 24.9433,C -1.7396,E1 25.145,E2 474.773} C_DIS
LIN {X 100.0297,Y -44.2871,Z 108,A -27.6039,B 24.9429,C -1.7448,E1 25.1466,E2 473.317} C_DIS
LIN {X 101.0865,Y -41.8189,Z 108,A -26.2812,B 24.9429,C -1.7454,E1 25.1481,E2 472.0003} C_DIS
LIN {X 102.0651,Y -39.3709,Z 108,A -24.8647,B 24.9425,C -1.7513,E1 25.1495,E2 470.5777} C_DIS
LIN {X 103.0006,Y -36.8542,Z 108,A -23.4897,B 24.9423,C -1.7543,E1 25.1508,E2 469.2033} C_DIS
LIN {X 103.874,Y -34.3153,Z 108,A -22.0933,B 24.9421,C -1.7583,E1 25.1521,E2 467.8054} C_DIS
LIN {X 104.7597,Y -31.5037,Z 108,A -20.6569,B 24.9421,C -1.7583,E1 25.1533,E2 466.3771} C_DIS
LIN {X 105.4453,Y -29.1303,Z 108,A -19.2975,B 24.9416,C -1.7654,E1 25.1543,E2 465.0089} C_DIS
LIN {X 106.117,Y -26.5809,Z 108,A -17.9031,B 24.9413,C -1.7704,E1 25.1553,E2 463.6106} C_DIS
LIN {X 106.7884,Y -23.7347,Z 108,A -16.4955,B 24.9413,C -1.7698,E1 25.1561,E2 462.2127} C_DIS
LIN {X 107.2934,Y -21.342,Z 108,A -14.9648,B 24.9403,C -1.7851,E1 25.157,E2 460.6548} C_DIS
LIN {X 107.7928,Y -18.6546,Z 108,A -13.7112,B 24.9405,C -1.7817,E1 25.1576,E2 459.4165} C_DIS
LIN {X 108.2528,Y -15.7603,Z 108,A -12.2751,B 24.9405,C -1.7823,E1 25.1582,E2 457.9875} C_DIS
LIN {X 108.5727,Y -13.3912,Z 108,A -10.9205,B 24.9399,C -1.7909,E1 25.1587,E2 456.6205} C_DIS
LIN {X 108.8731,Y -10.6743,Z 108,A -9.4989,B 24.9396,C -1.7951,E1 25.1591,E2 455.1975} C_DIS
LIN {X 109.099,Y -8.0476,Z 108,A -8.0647,B 24.9391,C -1.802,E1 25.1594,E2 453.7555} C_DIS
LIN {X 109.2636,Y -5.3678,Z 108,A -6.7091,B 24.939,C -1.8043,E1 25.1596,E2 452.4026} C_DIS
LIN {X 109.3625,Y -2.6847,Z 108,A -5.3349,B 24.9388,C -1.8074,E1 25.1598,E2 451.0293} C_DIS
LIN {X 109.3945,Y 0,Z 108,A -3.9506,B 24.9385,C -1.811,E1 25.1598,E2 449.6447} C_DIS
LIN {X 109.3625,Y 2.6847,Z 108,A -2.5197,B 24.9381,C -1.8167,E1 25.1598,E2 448.2089} C_DIS
LIN {X 109.2636,Y 5.3678,Z 108,A -1.1233,B 24.9379,C -1.8208,E1 25.1595,E2 446.8112} C_DIS
LIN {X 109.099,Y 8.0476,Z 108,A 0.2513,B 24.9376,C -1.8239,E1 25.1593,E2 445.4374} C_DIS
LIN {X 108.8636,Y 10.7708,Z 108,A 1.6729,B 24.9374,C -1.828,E1 25.1589,E2 444.0145} C_DIS
LIN {X 108.4966,Y 13.9782,Z 108,A 3.1107,B 24.9378,C -1.8221,E1 25.1584,E2 442.5991} C_DIS
LIN {X 108.204,Y 16.0996,Z 108,A 4.4663,B 24.9368,C -1.8361,E1 25.1579,E2 441.2185} C_DIS
LIN {X 107.7849,Y 18.7024,Z 108,A 5.8602,B 24.9365,C -1.8411,E1 25.1573,E2 439.8211} C_DIS
LIN {X 107.2934,Y 21.342,Z 108,A 7.2345,B 24.9363,C -1.8441,E1 25.1565,E2 438.4477} C_DIS
LIN {X 106.7373,Y 23.9687,Z 108,A 8.7182,B 24.9357,C -1.8519,E1 25.1556,E2 436.9542} C_DIS
LIN {X 106.117,Y 26.5809,Z 108,A 10.0283,B 24.9357,C -1.8519,E1 25.1548,E2 435.6515} C_DIS
LIN {X 105.4327,Y 29.1771,Z 108,A 11.5986,B 24.9349,C -1.8636,E1 25.1536,E2 434.0628} C_DIS
LIN {X 104.6705,Y 31.8021,Z 108,A 12.8245,B 24.9352,C -1.8588,E1 25.1526,E2 432.8552} C_DIS
LIN {X 103.7235,Y 34.7618,Z 108,A 14.2413,B 24.9355,C -1.8544,E1 25.1514,E2 431.4568} C_DIS
LIN {X 103.0006,Y 36.8542,Z 108,A 15.6392,B 24.9346,C -1.8684,E1 25.1501,E2 430.0338} C_DIS
LIN {X 102.0474,Y 39.416,Z 108,A 17.1216,B 24.9341,C -1.8749,E1 25.1486,E2 428.5443} C_DIS
LIN {X 101.0682,Y 41.8638,Z 108,A 18.4116,B 24.9341,C -1.8749,E1 25.1473,E2 427.2614} C_DIS
LIN {X 100.0104,Y 44.3315,Z 108,A 19.8314,B 24.9338,C -1.8795,E1 25.1457,E2 425.8383} C_DIS
LIN {X 98.8713,Y 46.8163,Z 108,A 21.232,B 24.9336,C -1.8822,E1 25.144,E2 424.4389} C_DIS
LIN {X 97.7146,Y 49.1854,Z 108,A 22.7872,B 24.9328,C -1.8938,E1 25.1421,E2 422.8647} C_DIS
LIN {X 96.455,Y 51.6113,Z 108,A 24.0047,B 24.9332,C -1.8883,E1 25.1405,E2 421.6666} C_DIS
LIN {X 95.1835,Y 53.9208,Z 108,A 25.4228,B 24.9328,C -1.8937,E1 25.1386,E2 420.2432} C_DIS
LIN {X 93.7364,Y 56.3971,Z 108,A 26.8326,B 24.9328,C -1.8937,E1 25.1366,E2 418.8406} C_DIS
LIN {X 92.3969,Y 58.5671,Z 108,A 28.2223,B 24.9324,C -1.8996,E1 25.1345,E2 417.4441} C_DIS
LIN {X 90.959,Y 60.7768,Z 108,A 29.5951,B 24.9321,C -1.9028,E1 25.1324,E2 416.0705} C_DIS
LIN {X 89.44,Y 62.9908,Z 108,A 31.0161,B 24.9318,C -1.907,E1 25.1301,E2 414.6466} C_DIS
LIN {X 87.7185,Y 65.3648,Z 108,A 32.4037,B 24.932,C -1.9044,E1 25.1279,E2 413.2718} C_DIS
LIN {X 86.2114,Y 67.3416,Z 108,A 33.7935,B 24.9315,C -1.9114,E1 25.1255,E2 411.872} C_DIS
LIN {X 84.5328,Y 69.437,Z 108,A 35.2156,B 24.9312,C -1.9154,E1 25.123,E2 410.447} C_DIS
LIN {X 82.541,Y 71.7909,Z 108,A 36.6431,B 24.9315,C -1.9111,E1 25.1204,E2 409.0364} C_DIS
LIN {X 81.0239,Y 73.5012,Z 108,A 37.9911,B 24.9309,C -1.9203,E1 25.1179,E2 407.6725} C_DIS
LIN {X 79.2293,Y 75.4326,Z 108,A 39.4111,B 24.9305,C -1.9251,E1 25.1151,E2 406.2475} C_DIS
LIN {X 77.3542,Y 77.3542,Z 108,A 40.7881,B 24.9304,C -1.9268,E1 25.1124,E2 404.8721} C_DIS
LIN {X 75.4326,Y 79.2293,Z 108,A 42.2231,B 24.9301,C -1.931,E1 25.1095,E2 403.4331} C_DIS
LIN {X 73.2697,Y 81.2319,Z 108,A 43.6279,B 24.9303,C -1.9282,E1 25.1067,E2 402.0408} C_DIS
LIN {X 71.4172,Y 82.8666,Z 108,A 45.0139,B 24.9298,C -1.9347,E1 25.1037,E2 400.6449} C_DIS
LIN {X 69.3997,Y 84.5638,Z 108,A 46.4114,B 24.9296,C -1.9381,E1 25.1007,E2 399.2448} C_DIS
LIN {X 66.2401,Y 87.0609,Z 108,A 48.4899,B 24.9294,C -1.9406,E1 25.0961,E2 397.1679} C_DIS
LIN {X 64.0441,Y 88.6885,Z 108,A 49.8931,B 24.9294,C -1.9419,E1 25.093,E2 395.7667} C_DIS
LIN {X 61.8483,Y 90.2335,Z 108,A 51.3174,B 24.9291,C -1.945,E1 25.0897,E2 394.3399} C_DIS
LIN {X 59.6561,Y 91.6979,Z 108,A 52.6937,B 24.9289,C -1.9471,E1 25.0865,E2 392.9634} C_DIS
LIN {X 57.3463,Y 93.1595,Z 108,A 54.1572,B 24.9287,C -1.9506,E1 25.083,E2 391.496} C_DIS
LIN {X 55.0848,Y 94.5147,Z 108,A 55.4969,B 24.9287,C -1.9509,E1 25.0798,E2 390.1597} C_DIS
LIN {X 52.7487,Y 95.838,Z 108,A 56.9212,B 24.9284,C -1.9537,E1 25.0763,E2 388.7332} C_DIS
LIN {X 50.3376,Y 97.1258,Z 108,A 58.4778,B 24.9279,C -1.9609,E1 25.0725,E2 387.1638} C_DIS
LIN {X 47.9389,Y 98.3319,Z 108,A 59.7056,B 24.9283,C -1.9551,E1 25.0694,E2 385.953} C_DIS
LIN {X 45.5555,Y 99.4588,Z 108,A 61.1283,B 24.9281,C -1.9585,E1 25.0658,E2 384.526} C_DIS
LIN {X 42.5724,Y 100.7696,Z 108,A 62.5733,B 24.9288,C -1.9494,E1 25.0622,E2 383.1059} C_DIS
LIN {X 40.6204,Y 101.5743,Z 108,A 63.9123,B 24.928,C -1.9603,E1 25.0586,E2 381.7442} C_DIS
LIN {X 37.9367,Y 102.6058,Z 108,A 65.324,B 24.9281,C -1.9578,E1 25.055,E2 380.3415} C_DIS
LIN {X 35.5093,Y 103.4715,Z 108,A 66.7602,B 24.9278,C -1.9626,E1 25.0512,E2 378.8968} C_DIS
LIN {X 33.0381,Y 104.2873,Z 108,A 68.1231,B 24.9278,C -1.9637,E1 25.0476,E2 377.5339} C_DIS
LIN {X 30.4221,Y 105.0799,Z 108,A 69.529,B 24.9278,C -1.9637,E1 25.0438,E2 376.1304} C_DIS
LIN {X 27.8342,Y 105.7949,Z 108,A 70.9544,B 24.9276,C -1.9654,E1 25.0399,E2 374.7032} C_DIS
LIN {X 25.2295,Y 106.4461,Z 108,A 72.3609,B 24.9276,C -1.9662,E1 25.0361,E2 373.2968} C_DIS
LIN {X 22.6095,Y 107.0332,Z 108,A 73.7427,B 24.9276,C -1.9659,E1 25.0324,E2 371.9176} C_DIS
LIN {X 20.0237,Y 107.5472,Z 108,A 75.1676,B 24.9274,C -1.9683,E1 25.0284,E2 370.4887} C_DIS
LIN {X 17.3784,Y 108.0062,Z 108,A 76.7006,B 24.9269,C -1.974,E1 25.0242,E2 368.9437} C_DIS
LIN {X 14.6744,Y 108.4064,Z 108,A 77.958,B 24.9274,C -1.9672,E1 25.0208,E2 367.7035} C_DIS
LIN {X 12.0578,Y 108.7289,Z 108,A 79.3618,B 24.9274,C -1.9684,E1 25.0169,E2 366.2979} C_DIS
LIN {X 8.8983,Y 109.031,Z 108,A 80.7899,B 24.9281,C -1.959,E1 25.013,E2 364.8929} C_DIS
LIN {X 6.6598,Y 109.1922,Z 108,A 82.2778,B 24.9271,C -1.9717,E1 25.0087,E2 363.3754} C_DIS
LIN {X 3.9781,Y 109.3228,Z 108,A 83.5825,B 24.9274,C -1.9675,E1 25.0051,E2 362.0811} C_DIS
LIN {X 1.1029,Y 109.3886,Z 108,A 85.025,B 24.9276,C -1.9647,E1 25.0011,E2 360.6455} C_DIS
LIN {X -1.3909,Y 109.3863,Z 108,A 86.3963,B 24.9275,C -1.9671,E1 24.9973,E2 359.2686} C_DIS
LIN {X -4.075,Y 109.3192,Z 108,A 87.8032,B 24.9275,C -1.9667,E1 24.9933,E2 357.8624} C_DIS
LIN {X -6.7566,Y 109.1863,Z 108,A 89.2819,B 24.9273,C -1.9691,E1 24.9892,E2 356.3776} C_DIS
LIN {X -9.8756,Y 108.9468,Z 108,A 90.6734,B 24.9281,C -1.9584,E1 24.9854,E2 355.0109} C_DIS
LIN {X -12.106,Y 108.7232,Z 108,A 92.026,B 24.9276,C -1.9649,E1 24.9816,E2 353.6419} C_DIS
LIN {X -14.7705,Y 108.3934,Z 108,A 93.4575,B 24.9276,C -1.9651,E1 24.9776,E2 352.209} C_DIS
LIN {X -17.3784,Y 108.0062,Z 108,A 94.8402,B 24.9276,C -1.9642,E1 24.9738,E2 350.8271} C_DIS
LIN {X -20.0713,Y 107.5381,Z 108,A 96.4208,B 24.9273,C -1.9691,E1 24.9694,E2 349.2332} C_DIS
LIN {X -22.7044,Y 107.0131,Z 108,A 97.6833,B 24.9278,C -1.9621,E1 24.966,E2 347.9858} C_DIS
LIN {X -25.6604,Y 106.3416,Z 108,A 99.0849,B 24.9285,C -1.9533,E1 24.9623,E2 346.6035} C_DIS
LIN {X -27.8811,Y 105.7828,Z 108,A 100.4761,B 24.928,C -1.9597,E1 24.9585,E2 345.195} C_DIS
LIN {X -30.5153,Y 105.0529,Z 108,A 101.9109,B 24.9281,C -1.9583,E1 24.9546,E2 343.7612} C_DIS
LIN {X -33.0842,Y 104.2724,Z 108,A 103.3207,B 24.9282,C -1.9568,E1 24.9508,E2 342.3525} C_DIS
LIN {X -35.9142,Y 103.3304,Z 108,A 104.721,B 24.9288,C -1.9485,E1 24.9472,E2 340.9692} C_DIS
LIN {X -38.1607,Y 102.5234,Z 108,A 106.1409,B 24.9284,C -1.9536,E1 24.9434,E2 339.5344} C_DIS
LIN {X -41.8638,Y 101.0682,Z 108,A 108.2311,B 24.9286,C -1.9509,E1 24.938,E2 337.4458} C_DIS
LIN {X -44.3315,Y 100.0104,Z 108,A 109.6644,B 24.9287,C -1.9499,E1 24.9343,E2 336.0115} C_DIS
LIN {X -46.7726,Y 98.8923,Z 108,A 111.0529,B 24.9289,C -1.9471,E1 24.9308,E2 334.6264} C_DIS
LIN {X -49.1854,Y 97.7146,Z 108,A 112.4637,B 24.9291,C -1.945,E1 24.9273,E2 333.2168} C_DIS
LIN {X -51.6113,Y 96.455,Z 108,A 113.9228,B 24.9291,C -1.9437,E1 24.9237,E2 331.7569} C_DIS
LIN {X -53.9628,Y 95.1594,Z 108,A 115.3124,B 24.9294,C -1.9405,E1 24.9203,E2 330.3707} C_DIS
LIN {X -56.2819,Y 93.8064,Z 108,A 116.7244,B 24.9296,C -1.9382,E1 24.9169,E2 328.96} C_DIS
LIN {X -59.0142,Y 92.1099,Z 108,A 118.1761,B 24.9305,C -1.926,E1 24.9136,E2 327.5326} C_DIS
LIN {X -60.817,Y 90.9318,Z 108,A 119.5485,B 24.9299,C -1.9333,E1 24.9103,E2 326.1385} C_DIS
LIN {X -62.9908,Y 89.44,Z 108,A 120.9578,B 24.9301,C -1.9316,E1 24.9071,E2 324.7284} C_DIS
LIN {X -65.2055,Y 87.8381,Z 108,A 122.3736,B 24.9303,C -1.928,E1 24.9039,E2 323.3161} C_DIS
LIN {X -67.3035,Y 86.2415,Z 108,A 123.7834,B 24.9304,C -1.9262,E1 24.9008,E2 321.9055} C_DIS
LIN {X -69.3997,Y 84.5638,Z 108,A 125.174,B 24.9307,C -1.9225,E1 24.8978,E2 320.5184} C_DIS
LIN {X -71.4541,Y 82.8352,Z 108,A 126.6093,B 24.9309,C -1.9205,E1 24.8947,E2 319.0823} C_DIS
LIN {X -73.5012,Y 81.0239,Z 108,A 128.0257,B 24.9311,C -1.9166,E1 24.8918,E2 317.6696} C_DIS
LIN {X -75.4675,Y 79.1957,Z 108,A 129.4389,B 24.9314,C -1.9136,E1 24.8889,E2 316.2579} C_DIS
LIN {X -77.3542,Y 77.3542,Z 108,A 130.8803,B 24.9314,C -1.9125,E1 24.886,E2 314.8127} C_DIS
LIN {X -79.2625,Y 75.3972,Z 108,A 132.243,B 24.9319,C -1.9064,E1 24.8834,E2 313.4588} C_DIS
LIN {X -81.089,Y 73.4293,Z 108,A 133.657,B 24.9321,C -1.9031,E1 24.8808,E2 312.0464} C_DIS
LIN {X -82.8352,Y 71.4541,Z 108,A 135.0723,B 24.9323,C -1.9009,E1 24.8782,E2 310.63} C_DIS
LIN {X -84.5943,Y 69.362,Z 108,A 136.5085,B 24.9325,C -1.8973,E1 24.8756,E2 309.1957} C_DIS
LIN {X -86.2711,Y 67.2651,Z 108,A 137.923,B 24.9328,C -1.8939,E1 24.8731,E2 307.7827} C_DIS
LIN {X -87.8672,Y 65.1668,Z 108,A 139.3344,B 24.9329,C -1.8913,E1 24.8708,E2 306.3706} C_DIS
LIN {X -89.44,Y 62.9908,Z 108,A 140.7268,B 24.9333,C -1.8869,E1 24.8685,E2 304.9818} C_DIS
LIN {X -90.975,Y 60.7525,Z 108,A 142.1657,B 24.9335,C -1.8836,E1 24.8663,E2 303.5436} C_DIS
LIN {X -92.4231,Y 58.5263,Z 108,A 143.5787,B 24.9337,C -1.8805,E1 24.8642,E2 302.1309} C_DIS
LIN {X -93.8562,Y 56.1987,Z 108,A 144.9971,B 24.934,C -1.8759,E1 24.8621,E2 300.7162} C_DIS
LIN {X -95.2072,Y 53.8785,Z 108,A 146.3888,B 24.9344,C -1.8713,E1 24.8602,E2 299.3283} C_DIS
LIN {X -96.4781,Y 51.5686,Z 108,A 147.8018,B 24.9346,C -1.8685,E1 24.8583,E2 297.9146} C_DIS
LIN {X -97.7146,Y 49.1854,Z 108,A 149.2398,B 24.9348,C -1.8655,E1 24.8565,E2 296.476} C_DIS
LIN {X -98.8923,Y 46.7726,Z 108,A 150.6327,B 24.9351,C -1.8608,E1 24.8548,E2 295.0869} C_DIS
LIN {X -100.0297,Y 44.2871,Z 108,A 152.0738,B 24.9354,C -1.8568,E1 24.8531,E2 293.6474} C_DIS
LIN {X -101.0682,Y 41.8638,Z 108,A 153.4639,B 24.9356,C -1.8529,E1 24.8516,E2 292.2588} C_DIS
LIN {X -102.0651,Y 39.3709,Z 108,A 154.9018,B 24.9359,C -1.8498,E1 24.8502,E2 290.8203} C_DIS
LIN {X -103.0167,Y 36.8084,Z 108,A 156.3207,B 24.9362,C -1.8448,E1 24.8488,E2 289.4051} C_DIS
LIN {X -103.889,Y 34.2692,Z 108,A 157.7131,B 24.9365,C -1.8399,E1 24.8476,E2 288.0164} C_DIS
LIN {X -104.6849,Y 31.7558,Z 108,A 159.1493,B 24.9367,C -1.8377,E1 24.8464,E2 286.5775} C_DIS
LIN {X -105.4453,Y 29.1303,Z 108,A 160.545,B 24.9371,C -1.8318,E1 24.8453,E2 285.1876} C_DIS
LIN {X -106.117,Y 26.5809,Z 108,A 161.9589,B 24.9373,C -1.8286,E1 24.8444,E2 283.7731} C_DIS
LIN {X -106.7981,Y 23.6901,Z 108,A 163.4163,B 24.9379,C -1.82,E1 24.8435,E2 282.3277} C_DIS
LIN {X -107.2934,Y 21.342,Z 108,A 164.867,B 24.9377,C -1.8232,E1 24.8426,E2 280.8607} C_DIS
LIN {X -107.7849,Y 18.7024,Z 108,A 166.2071,B 24.9382,C -1.8162,E1 24.842,E2 279.5294} C_DIS
LIN {X -108.2182,Y 16.0036,Z 108,A 167.6487,B 24.9385,C -1.812,E1 24.8414,E2 278.0893} C_DIS
LIN {X -108.5727,Y 13.3912,Z 108,A 169.0394,B 24.9387,C -1.8079,E1 24.8409,E2 276.7001} C_DIS
LIN {X -108.8731,Y 10.6743,Z 108,A 170.481,B 24.939,C -1.8036,E1 24.8405,E2 275.26} C_DIS
LIN {X -109.099,Y 8.0476,Z 108,A 171.8942,B 24.9392,C -1.8004,E1 24.8401,E2 273.8461} C_DIS
LIN {X -109.2636,Y 5.3678,Z 108,A 173.3102,B 24.9395,C -1.7962,E1 24.8399,E2 272.4315} C_DIS
LIN {X -109.3625,Y 2.6847,Z 108,A 174.73,B 24.9398,C -1.7921,E1 24.8399,E2 271.0129} C_DIS
LIN {X -109.3945,Y 0,Z 108,A 176.1075,B 24.9402,C -1.7865,E1 24.8398,E2 269.6404} C_DIS
LIN {X -109.3625,Y -2.6847,Z 108,A 177.5586,B 24.9404,C -1.7836,E1 24.8398,E2 268.1874} C_DIS
LIN {X -109.2636,Y -5.3678,Z 108,A 178.9746,B 24.9406,C -1.7795,E1 24.84,E2 266.7728} C_DIS
LIN {X -109.099,Y -8.0476,Z 108,A -179.6313,B 24.941,C -1.7745,E1 24.8403,E2 265.3822} C_DIS
LIN {X -108.8636,Y -10.7708,Z 108,A -178.0613,B 24.941,C -1.7752,E1 24.8407,E2 263.8011} C_DIS
LIN {X -108.5727,Y -13.3912,Z 108,A -176.777,B 24.9415,C -1.7671,E1 24.8411,E2 262.5284} C_DIS
LIN {X -108.204,Y -16.0996,Z 108,A -175.3814,B 24.9419,C -1.7612,E1 24.8417,E2 261.1386} C_DIS
LIN {X -107.7849,Y -18.7024,Z 108,A -173.9451,B 24.942,C -1.759,E1 24.8423,E2 259.6991} C_DIS
LIN {X -107.2837,Y -21.3895,Z 108,A -172.5265,B 24.9423,C -1.754,E1 24.8431,E2 258.284} C_DIS
LIN {X -106.7264,Y -24.0159,Z 108,A -171.1105,B 24.9426,C -1.75,E1 24.8439,E2 256.8692} C_DIS
LIN {X -106.1049,Y -26.6279,Z 108,A -169.7183,B 24.9429,C -1.7451,E1 24.8449,E2 255.4805} C_DIS
LIN {X -105.4327,Y -29.1772,Z 108,A -168.3047,B 24.9431,C -1.7421,E1 24.8459,E2 254.0658} C_DIS
LIN {X -104.6705,Y -31.8021,Z 108,A -166.6891,B 24.9429,C -1.7448,E1 24.8472,E2 252.4345} C_DIS
LIN {X -103.8585,Y -34.3613,Z 108,A -165.448,B 24.9436,C -1.7342,E1 24.8483,E2 251.2114} C_DIS
LIN {X -103.0006,Y -36.8542,Z 108,A -164.0358,B 24.9438,C -1.7313,E1 24.8496,E2 249.7981} C_DIS
LIN {X -102.0474,Y -39.416,Z 108,A -162.6409,B 24.9442,C -1.7257,E1 24.8509,E2 248.4088} C_DIS
LIN {X -101.0682,Y -41.8638,Z 108,A -161.228,B 24.9444,C -1.7229,E1 24.8524,E2 246.9947} C_DIS
LIN {X -100.0104,Y -44.3315,Z 108,A -159.7903,B 24.9446,C -1.7201,E1 24.854,E2 245.5559} C_DIS
LIN {X -98.8923,Y -46.7726,Z 108,A -158.2345,B 24.9444,C -1.7218,E1 24.8559,E2 243.9874} C_DIS
LIN {X -97.6074,Y -49.3953,Z 108,A -156.9726,B 24.9454,C -1.7073,E1 24.8574,E2 242.7534} C_DIS
LIN {X -96.455,Y -51.6113,Z 108,A -155.5666,B 24.9454,C -1.7074,E1 24.8593,E2 241.3396} C_DIS
LIN {X -95.1835,Y -53.9208,Z 108,A -154.1314,B 24.9454,C -1.7057,E1 24.8612,E2 239.9008} C_DIS
LIN {X -93.8064,Y -56.2819,Z 108,A -152.7139,B 24.9458,C -1.7014,E1 24.8633,E2 238.4864} C_DIS
LIN {X -92.2569,Y -58.7852,Z 108,A -151.2821,B 24.9463,C -1.6931,E1 24.8654,E2 237.067} C_DIS
LIN {X -90.959,Y -60.7768,Z 108,A -149.8886,B 24.9461,C -1.6956,E1 24.8675,E2 235.6606} C_DIS
LIN {X -89.43,Y -63.0049,Z 108,A -148.4962,B 24.9464,C -1.6911,E1 24.8697,E2 234.272} C_DIS
LIN {X -87.8672,Y -65.1668,Z 108,A -147.0833,B 24.9466,C -1.6883,E1 24.8721,E2 232.859} C_DIS
LIN {X -86.2415,Y -67.3035,Z 108,A -145.6472,B 24.9467,C -1.686,E1 24.8745,E2 231.4215} C_DIS
LIN {X -84.3679,Y -69.6354,Z 108,A -144.2418,B 24.9474,C -1.6761,E1 24.877,E2 230.0332} C_DIS
LIN {X -82.8352,Y -71.4541,Z 108,A -142.8203,B 24.9471,C -1.68,E1 24.8796,E2 228.5959} C_DIS
LIN {X -80.149,Y -74.4546,Z 108,A -140.5402,B 24.947,C -1.682,E1 24.8839,E2 226.301} C_DIS
LIN {X -78.2636,Y -76.4337,Z 108,A -139.1337,B 24.9472,C -1.6779,E1 24.8866,E2 224.8982} C_DIS
LIN {X -76.3992,Y -78.2977,Z 108,A -137.8753,B 24.9477,C -1.6701,E1 24.8891,E2 223.6529} C_DIS
LIN {X -74.4546,Y -80.149,Z 108,A -136.2911,B 24.9475,C -1.6743,E1 24.8924,E2 222.0525} C_DIS
LIN {X -72.4287,Y -81.984,Z 108,A -135.0474,B 24.9481,C -1.664,E1 24.8949,E2 220.8282} C_DIS
LIN {X -70.3311,Y -83.7899,Z 108,A -133.6546,B 24.9484,C -1.659,E1 24.8979,E2 219.442} C_DIS
LIN {X -68.3187,Y -85.4391,Z 108,A -132.2233,B 24.9484,C -1.6591,E1 24.901,E2 218.0049} C_DIS
LIN {X -66.2014,Y -87.09,Z 108,A -130.8115,B 24.9486,C -1.6568,E1 24.9041,E2 216.5934} C_DIS
LIN {X -64.0441,Y -88.6885,Z 108,A -129.4233,B 24.9488,C -1.6537,E1 24.9072,E2 215.2078} C_DIS
LIN {X -61.8483,Y -90.2335,Z 108,A -128.0121,B 24.9488,C -1.6516,E1 24.9105,E2 213.7969} C_DIS
LIN {X -59.6152,Y -91.7241,Z 108,A -126.6007,B 24.949,C -1.6495,E1 24.9137,E2 212.3857} C_DIS
LIN {X -57.3877,Y -93.1343,Z 108,A -125.1924,B 24.949,C -1.6485,E1 24.9171,E2 210.9754} C_DIS
LIN {X -55.0427,Y -94.5388,Z 108,A -123.5905,B 24.9488,C -1.6533,E1 24.921,E2 209.3573} C_DIS
LIN {X -51.5257,Y -96.5007,Z 108,A -121.641,B 24.9494,C -1.644,E1 24.9257,E2 207.4243} C_DIS
LIN {X -49.142,Y -97.7362,Z 108,A -120.2306,B 24.9494,C -1.6424,E1 24.9292,E2 206.0139} C_DIS
LIN {X -46.7726,Y -98.8923,Z 108,A -118.7535,B 24.9494,C -1.6446,E1 24.933,E2 204.5278} C_DIS
LIN {X -43.9771,Y -100.1649,Z 108,A -117.3872,B 24.95,C -1.6331,E1 24.9364,E2 203.1856} C_DIS
LIN {X -41.8189,Y -101.0865,Z 108,A -116.0246,B 24.9498,C -1.6372,E1 24.9399,E2 201.8101} C_DIS
LIN {X -39.3709,Y -102.0651,Z 108,A -114.5955,B 24.9498,C -1.6378,E1 24.9437,E2 200.3765} C_DIS
LIN {X -36.8542,Y -103.0006,Z 108,A -113.2086,B 24.9498,C -1.6357,E1 24.9473,E2 198.9916} C_DIS
LIN {X -34.3153,Y -103.874,Z 108,A -111.8002,B 24.9499,C -1.6347,E1 24.951,E2 197.5831} C_DIS
LIN {X -31.7093,Y -104.6987,Z 108,A -110.3662,B 24.9499,C -1.6337,E1 24.9548,E2 196.1489} C_DIS
LIN {X -29.1303,Y -105.4453,Z 108,A -108.9811,B 24.9501,C -1.6319,E1 24.9586,E2 194.7659} C_DIS
LIN {X -26.5809,Y -106.117,Z 108,A -107.5753,B 24.9501,C -1.6322,E1 24.9624,E2 193.3574} C_DIS
LIN {X -23.9687,Y -106.7373,Z 108,A -106.1676,B 24.9501,C -1.6315,E1 24.9662,E2 191.9495} C_DIS
LIN {X -21.342,Y -107.2934,Z 108,A -104.7377,B 24.9501,C -1.6319,E1 24.9701,E2 190.517} C_DIS
LIN {X -18.6546,Y -107.7928,Z 108,A -103.3504,B 24.9502,C -1.6296,E1 24.9739,E2 189.1338} C_DIS
LIN {X -16.0516,Y -108.2114,Z 108,A -101.9234,B 24.9502,C -1.6311,E1 24.9779,E2 187.7018} C_DIS
LIN {X -13.3912,Y -108.5727,Z 108,A -100.5388,B 24.9502,C -1.63,E1 24.9817,E2 186.319} C_DIS
LIN {X -10.6743,Y -108.8731,Z 108,A -98.9569,B 24.9498,C -1.6361,E1 24.9861,E2 184.7217} C_DIS
LIN {X -8.0476,Y -109.099,Z 108,A -97.7036,B 24.9502,C -1.6307,E1 24.9896,E2 183.4805} C_DIS
LIN {X -5.3678,Y -109.2636,Z 108,A -96.243,B 24.95,C -1.6331,E1 24.9937,E2 182.014} C_DIS
LIN {X -2.6847,Y -109.3625,Z 108,A -94.9143,B 24.9502,C -1.63,E1 24.9974,E2 180.6923} C_DIS
LIN {X 0.0485,Y -109.3951,Z 108,A -93.4833,B 24.9502,C -1.6303,E1 25.0014,E2 179.2607} C_DIS
LIN {X 0.0485,Y -109.3951,Z 108,A -93.4833,B 24.9502,C -1.6303,E1 25.0014,E2 179.2607} C_DIS
Enddeposition()
LIN {X 0.7534,Y -108.4284,Z 108,A -93.4914,B 24.9502,C -1.6315,E1 25.0014,E2 179.2659} C_DIS
Startdeposition()
$VEL.CP = VEL_PRINT
LIN {X -1.9035,Y -108.4187,Z 108,A -95.3707,B 24.9513,C -1.6117,E1 24.996,E2 181.1923} C_DIS
LIN {X -5.2751,Y -108.3087,Z 108,A -96.9649,B 24.9509,C -1.6191,E1 24.9916,E2 182.7691} C_DIS
LIN {X -7.9878,Y -108.1425,Z 108,A -98.4213,B 24.9509,C -1.6183,E1 24.9875,E2 184.228} C_DIS
LIN {X -10.4435,Y -107.9323,Z 108,A -99.7132,B 24.9509,C -1.6188,E1 24.9839,E2 185.5194} C_DIS
LIN {X -12.7269,Y -107.6859,Z 108,A -101.0045,B 24.9511,C -1.6158,E1 24.9803,E2 186.8185} C_DIS
LIN {X -16.8347,Y -107.1209,Z 108,A -103.2354,B 24.9511,C -1.6147,E1 24.9741,E2 189.0538} C_DIS
LIN {X -20.6982,Y -106.4418,Z 108,A -105.2245,B 24.9509,C -1.6188,E1 24.9687,E2 191.0353} C_DIS
LIN {X -23.8141,Y -105.7898,Z 108,A -107.4026,B 24.952,C -1.5998,E1 24.9626,E2 193.2613} C_DIS
LIN {X -27.1308,Y -104.9865,Z 108,A -108.2908,B 24.9498,C -1.6374,E1 24.9605,E2 194.0615} C_DIS
LIN {X -29.6388,Y -104.3062,Z 108,A -111.2813,B 24.9536,C -1.5742,E1 24.952,E2 197.2068} C_DIS
LIN {X -35.7459,Y -102.3742,Z 108,A -113.5014,B 24.9507,C -1.6227,E1 24.9464,E2 199.316} C_DIS
LIN {X -38.9589,Y -101.1967,Z 108,A -115.2513,B 24.9504,C -1.6266,E1 24.9419,E2 201.0601} C_DIS
LIN {X -41.5289,Y -100.1696,Z 108,A -116.8662,B 24.9507,C -1.6221,E1 24.9377,E2 202.6895} C_DIS
LIN {X -44.6135,Y -98.8325,Z 108,A -118.5885,B 24.9504,C -1.6262,E1 24.9333,E2 204.4061} C_DIS
LIN {X -48.1155,Y -97.1757,Z 108,A -120.6445,B 24.9504,C -1.6283,E1 24.9281,E2 206.4624} C_DIS
LIN {X -51.5549,Y -95.3957,Z 108,A -122.6792,B 24.9501,C -1.6314,E1 24.9231,E2 208.4953} C_DIS
LIN {X -54.5673,Y -93.7071,Z 108,A -124.6472,B 24.9503,C -1.6284,E1 24.9183,E2 210.4763} C_DIS
LIN {X -57.7163,Y -91.7995,Z 108,A -126.4231,B 24.9497,C -1.6379,E1 24.9141,E2 212.2352} C_DIS
LIN {X -60.494,Y -89.9935,Z 108,A -128.26,B 24.9497,C -1.6374,E1 24.9098,E2 214.0794} C_DIS
LIN {X -63.392,Y -87.9769,Z 108,A -130.2567,B 24.9499,C -1.6354,E1 24.9052,E2 216.0876} C_DIS
LIN {X -66.0944,Y -85.9637,Z 108,A -131.8856,B 24.9493,C -1.6445,E1 24.9016,E2 217.7008} C_DIS
LIN {X -68.3831,Y -84.1546,Z 108,A -133.6051,B 24.9496,C -1.6405,E1 24.8979,E2 219.4363} C_DIS
LIN {X -70.7602,Y -82.1678,Z 108,A -135.0944,B 24.949,C -1.6493,E1 24.8947,E2 220.9105} C_DIS
LIN {X -73.1872,Y -80.0118,Z 108,A -136.7936,B 24.9488,C -1.6533,E1 24.8912,E2 222.6068} C_DIS
LIN {X -76.2849,Y -77.0639,Z 108,A -138.7009,B 24.9476,C -1.6715,E1 24.8874,E2 224.4787} C_DIS
LIN {X -78.1768,Y -75.1441,Z 108,A -140.4456,B 24.9482,C -1.6623,E1 24.884,E2 226.2528} C_DIS
LIN {X -80.5858,Y -72.5551,Z 108,A -142.2041,B 24.9477,C -1.6707,E1 24.8807,E2 227.9992} C_DIS
LIN {X -82.84,Y -69.9712,Z 108,A -144.1202,B 24.9477,C -1.6709,E1 24.8772,E2 229.9234} C_DIS
LIN {X -84.7653,Y -67.6263,Z 108,A -145.9814,B 24.9481,C -1.6649,E1 24.8739,E2 231.8076} C_DIS
LIN {X -87.7828,Y -63.6604,Z 108,A -148.3823,B 24.9471,C -1.6801,E1 24.8699,E2 234.1837} C_DIS
LIN {X -89.3646,Y -61.4209,Z 108,A -149.8226,B 24.9469,C -1.6841,E1 24.8676,E2 235.6216} C_DIS
LIN {X -90.6815,Y -59.4573,Z 108,A -151.4079,B 24.9474,C -1.6747,E1 24.8651,E2 237.2373} C_DIS
LIN {X -92.3817,Y -56.7816,Z 108,A -152.9367,B 24.9468,C -1.6846,E1 24.8629,E2 238.7504} C_DIS
LIN {X -94.3018,Y -53.5324,Z 108,A -154.8266,B 24.9462,C -1.6938,E1 24.8602,E2 240.6281} C_DIS
LIN {X -96.2468,Y -49.952,Z 108,A -156.9463,B 24.9458,C -1.701,E1 24.8575,E2 242.7419} C_DIS
LIN {X -97.3746,Y -47.7142,Z 108,A -158.2831,B 24.9456,C -1.7042,E1 24.8558,E2 244.0782} C_DIS
LIN {X -98.5496,Y -45.2387,Z 108,A -159.736,B 24.9453,C -1.7081,E1 24.8541,E2 245.5297} C_DIS
LIN {X -100.2095,Y -41.4323,Z 108,A -161.9176,B 24.9449,C -1.7149,E1 24.8517,E2 247.7072} C_DIS
LIN {X -101.3452,Y -38.5669,Z 108,A -163.7117,B 24.9449,C -1.7136,E1 24.8498,E2 249.5146} C_DIS
LIN {X -102.991,Y -33.9326,Z 108,A -166.1593,B 24.9441,C -1.7269,E1 24.8476,E2 251.9443} C_DIS
LIN {X -103.9579,Y -30.8381,Z 108,A -168.0245,B 24.9441,C -1.7265,E1 24.8461,E2 253.8213} C_DIS
LIN {X -104.7904,Y -27.8812,Z 108,A -169.5599,B 24.9436,C -1.7347,E1 24.845,E2 255.3461} C_DIS
LIN {X -105.617,Y -24.5619,Z 108,A -171.419,B 24.9434,C -1.7384,E1 24.8437,E2 257.2073} C_DIS
LIN {X -106.2844,Y -21.4929,Z 108,A -173.2534,B 24.9434,C -1.7371,E1 24.8427,E2 259.0556} C_DIS
LIN {X -107.0289,Y -17.4143,Z 108,A -175.2411,B 24.9425,C -1.7514,E1 24.8417,E2 261.0208} C_DIS
LIN {X -107.4084,Y -14.8926,Z 108,A -176.7575,B 24.9426,C -1.7495,E1 24.8411,E2 262.5508} C_DIS
LIN {X -107.8449,Y -11.3,Z 108,A -179.4641,B 24.9441,C -1.7266,E1 24.8403,E2 265.3283} C_DIS
LIN {X -108.2597,Y -6.1724,Z 108,A 178.9561,B 24.9408,C -1.777,E1 24.84,E2 266.7973} C_DIS
LIN {X -108.4343,Y -0.3986,Z 108,A 175.6339,B 24.9408,C -1.7768,E1 24.8398,E2 270.14} C_DIS
LIN {X -108.3937,Y 3.0216,Z 108,A 173.6374,B 24.9409,C -1.7757,E1 24.8398,E2 272.1512} C_DIS
LIN {X -108.2065,Y 7.0462,Z 108,A 171.1878,B 24.9412,C -1.7709,E1 24.8403,E2 274.6271} C_DIS
LIN {X -107.93,Y 10.4685,Z 108,A 169.8633,B 24.9396,C -1.7946,E1 24.8406,E2 275.9028} C_DIS
LIN {X -107.0097,Y 17.5293,Z 108,A 166.219,B 24.9385,C -1.8111,E1 24.842,E2 279.5296} C_DIS
LIN {X -106.171,Y 22.0452,Z 108,A 163.7341,B 24.9381,C -1.8168,E1 24.8433,E2 282.0157} C_DIS
LIN {X -105.635,Y 24.4841,Z 108,A 162.2218,B 24.9383,C -1.8139,E1 24.8442,E2 283.5438} C_DIS
LIN {X -104.8956,Y 27.4843,Z 108,A 160.666,B 24.9378,C -1.8219,E1 24.8453,E2 285.0896} C_DIS
LIN {X -104.3085,Y 29.6306,Z 108,A 159.5221,B 24.9374,C -1.8268,E1 24.8461,E2 286.2284} C_DIS
LIN {X -103.6616,Y 31.821,Z 108,A 158.1583,B 24.9376,C -1.8248,E1 24.8472,E2 287.6047} C_DIS
LIN {X -102.6423,Y 34.97,Z 108,A 156.5228,B 24.9369,C -1.8345,E1 24.8487,E2 289.2266} C_DIS
LIN {X -101.8975,Y 37.0829,Z 108,A 155.3516,B 24.9366,C -1.8386,E1 24.8498,E2 290.3945} C_DIS
LIN {X -100.8719,Y 39.7883,Z 108,A 153.3905,B 24.9374,C -1.8274,E1 24.8518,E2 292.3933} C_DIS
LIN {X -99.1016,Y 44.0163,Z 108,A 150.7908,B 24.9374,C -1.8283,E1 24.8547,E2 295.0053} C_DIS
LIN {X -97.6565,Y 47.1325,Z 108,A 148.9933,B 24.9369,C -1.8344,E1 24.8569,E2 296.798} C_DIS
LIN {X -96.1159,Y 50.2006,Z 108,A 147.524,B 24.9357,C -1.8524,E1 24.8587,E2 298.2322} C_DIS
LIN {X -94.4346,Y 53.297,Z 108,A 145.8158,B 24.9349,C -1.8635,E1 24.861,E2 299.9229} C_DIS
LIN {X -93.34,Y 55.1894,Z 108,A 144.7014,B 24.9346,C -1.8684,E1 24.8626,E2 301.0314} C_DIS
LIN {X -91.8596,Y 57.6201,Z 108,A 143.1354,B 24.9344,C -1.8704,E1 24.8649,E2 302.6007} C_DIS
LIN {X -90.1287,Y 60.2943,Z 108,A 141.4574,B 24.9341,C -1.8753,E1 24.8674,E2 304.2754} C_DIS
LIN {X -88.6568,Y 62.4391,Z 108,A 140.0454,B 24.9339,C -1.8777,E1 24.8697,E2 305.6886} C_DIS
LIN {X -87.2764,Y 64.352,Z 108,A 137.8726,B 24.9361,C -1.8469,E1 24.8734,E2 307.9452} C_DIS
LIN {X -84.1594,Y 68.3772,Z 108,A 136.4723,B 24.9322,C -1.9019,E1 24.8757,E2 309.2212} C_DIS
LIN {X -79.6793,Y 73.5496,Z 108,A 131.8821,B 24.9341,C -1.8747,E1 24.8843,E2 313.8967} C_DIS
LIN {X -77.1658,Y 76.1818,Z 108,A 130.824,B 24.9315,C -1.9118,E1 24.8862,E2 314.8711} C_DIS
LIN {X -74.3586,Y 78.9242,Z 108,A 128.4092,B 24.932,C -1.9039,E1 24.8911,E2 317.3148} C_DIS
LIN {X -71.1348,Y 81.8421,Z 108,A 125.5083,B 24.9333,C -1.8866,E1 24.8972,E2 320.2684} C_DIS
LIN {X -68.1865,Y 84.3139,Z 108,A 124.036,B 24.9315,C -1.9121,E1 24.9003,E2 321.6856} C_DIS
LIN {X -65.3407,Y 86.5384,Z 108,A 121.8551,B 24.9319,C -1.9058,E1 24.9052,E2 323.8893} C_DIS
LIN {X -59.6655,Y 90.5442,Z 108,A 118.3832,B 24.9308,C -1.9207,E1 24.9131,E2 327.3375} C_DIS
LIN {X -56.3406,Y 92.6497,Z 108,A 116.3802,B 24.9303,C -1.9275,E1 24.9178,E2 329.3307} C_DIS
LIN {X -53.3922,Y 94.3814,Z 108,A 114.4454,B 24.9305,C -1.9258,E1 24.9225,E2 331.2752} C_DIS
LIN {X -50.1711,Y 96.1314,Z 108,A 112.4397,B 24.9305,C -1.9265,E1 24.9275,E2 333.2849} C_DIS
LIN {X -46.3157,Y 98.0483,Z 108,A 109.9509,B 24.9308,C -1.9219,E1 24.9338,E2 335.791} C_DIS
LIN {X -42.9106,Y 99.5847,Z 108,A 108.1479,B 24.9301,C -1.9314,E1 24.9383,E2 337.5758} C_DIS
LIN {X -39.0716,Y 101.1534,Z 108,A 106.1794,B 24.9292,C -1.943,E1 24.9434,E2 339.5211} C_DIS
LIN {X -36.5878,Y 102.078,Z 108,A 104.5796,B 24.9297,C -1.9371,E1 24.9476,E2 341.1381} C_DIS
LIN {X -31.928,Y 103.6285,Z 108,A 102.166,B 24.9289,C -1.9472,E1 24.954,E2 343.532} C_DIS
LIN {X -29.0336,Y 104.4776,Z 108,A 100.3621,B 24.9294,C -1.9407,E1 24.9589,E2 345.3542} C_DIS
LIN {X -22.7856,Y 106.0149,Z 108,A 97.1673,B 24.9286,C -1.9519,E1 24.9675,E2 348.5268} C_DIS
LIN {X -19.6495,Y 106.6412,Z 108,A 94.6209,B 24.9309,C -1.9199,E1 24.9747,E2 351.1519} C_DIS
LIN {X -14.9152,Y 107.4052,Z 108,A 92.7915,B 24.9288,C -1.949,E1 24.9796,E2 352.9136} C_DIS
LIN {X -9.7846,Y 107.9931,Z 108,A 90.6033,B 24.9271,C -1.9719,E1 24.9855,E2 355.0489} C_DIS
LIN {X -5.4801,Y 108.298,Z 108,A 87.8463,B 24.9284,C -1.9538,E1 24.9933,E2 357.8498} C_DIS
LIN {X -1.1579,Y 108.4303,Z 108,A 85.3511,B 24.929,C -1.9461,E1 25.0003,E2 360.3635} C_DIS
LIN {X 3.369,Y 108.383,Z 108,A 83.143,B 24.9284,C -1.9538,E1 25.0064,E2 362.5531} C_DIS
LIN {X 6.2585,Y 108.2549,Z 108,A 81.5995,B 24.9284,C -1.9532,E1 25.0107,E2 364.0974} C_DIS
LIN {X 9.7272,Y 107.9984,Z 108,A 79.781,B 24.9284,C -1.9539,E1 25.0158,E2 365.9133} C_DIS
LIN {X 14.2235,Y 107.4988,Z 108,A 77.4166,B 24.9284,C -1.9544,E1 25.0223,E2 368.2746} C_DIS
LIN {X 18.0947,Y 106.9152,Z 108,A 75.2976,B 24.9286,C -1.9518,E1 25.0282,E2 370.3979} C_DIS
LIN {X 23.8862,Y 105.7731,Z 108,A 72.272,B 24.9284,C -1.9541,E1 25.0365,E2 373.4142} C_DIS
LIN {X 28.3006,Y 104.6771,Z 108,A 69.9133,B 24.9284,C -1.9545,E1 25.0428,E2 375.7685} C_DIS
LIN {X 32.1011,Y 103.5748,Z 108,A 67.7953,B 24.9286,C -1.9518,E1 25.0485,E2 377.889} C_DIS
LIN {X 35.2495,Y 102.548,Z 108,A 66.0603,B 24.9286,C -1.951,E1 25.0531,E2 379.6228} C_DIS
LIN {X 37.9204,Y 101.59,Z 108,A 64.6336,B 24.9286,C -1.9526,E1 25.0568,E2 381.0428} C_DIS
LIN {X 40.5025,Y 100.588,Z 108,A 62.969,B 24.9292,C -1.9428,E1 25.0612,E2 382.7267} C_DIS
LIN {X 43.8884,Y 99.1584,Z 108,A 60.982,B 24.9295,C -1.9388,E1 25.0663,E2 384.7184} C_DIS
LIN {X 47.4024,Y 97.5268,Z 108,A 59.0068,B 24.9295,C -1.9393,E1 25.0713,E2 386.6873} C_DIS
LIN {X 51.0292,Y 95.6795,Z 108,A 56.8231,B 24.9298,C -1.9351,E1 25.0767,E2 388.8749} C_DIS
LIN {X 53.4662,Y 94.3398,Z 108,A 55.3173,B 24.9301,C -1.9315,E1 25.0804,E2 390.3847} C_DIS
LIN {X 56.7353,Y 92.4098,Z 108,A 53.5429,B 24.9296,C -1.9382,E1 25.0846,E2 392.1379} C_DIS
LIN {X 59.1648,Y 90.8743,Z 108,A 52.0177,B 24.9298,C -1.9355,E1 25.0881,E2 393.6645} C_DIS
LIN {X 61.643,Y 89.2102,Z 108,A 50.3864,B 24.9301,C -1.9306,E1 25.0919,E2 395.3017} C_DIS
LIN {X 64.2548,Y 87.3476,Z 108,A 48.7392,B 24.9301,C -1.9297,E1 25.0956,E2 396.9453} C_DIS
LIN {X 66.8335,Y 85.3918,Z 108,A 47.1088,B 24.9301,C -1.9299,E1 25.0992,E2 398.5692} C_DIS
LIN {X 69.1238,Y 83.5475,Z 108,A 45.4578,B 24.9307,C -1.9229,E1 25.1028,E2 400.2305} C_DIS
LIN {X 71.958,Y 81.1204,Z 108,A 43.3567,B 24.9314,C -1.9136,E1 25.1073,E2 402.3455} C_DIS
LIN {X 74.8338,Y 78.4759,Z 108,A 41.315,B 24.9316,C -1.9102,E1 25.1115,E2 404.3866} C_DIS
LIN {X 77.3531,Y 75.9922,Z 108,A 39.4199,B 24.932,C -1.9052,E1 25.1152,E2 406.2858} C_DIS
LIN {X 80.0641,Y 73.1302,Z 108,A 37.6082,B 24.9315,C -1.9121,E1 25.1186,E2 408.0732} C_DIS
LIN {X 82.054,Y 70.8922,Z 108,A 35.7571,B 24.9325,C -1.8969,E1 25.1221,E2 409.9517} C_DIS
LIN {X 84.6526,Y 67.7686,Z 108,A 33.596,B 24.933,C -1.8912,E1 25.1259,E2 412.1163} C_DIS
LIN {X 87.0038,Y 64.7211,Z 108,A 31.8012,B 24.9326,C -1.8965,E1 25.1289,E2 413.8902} C_DIS
LIN {X 89.1344,Y 61.752,Z 108,A 29.8387,B 24.933,C -1.8902,E1 25.1321,E2 415.8578} C_DIS
LIN {X 91.1915,Y 58.6716,Z 108,A 27.8072,B 24.9336,C -1.882,E1 25.1352,E2 417.8987} C_DIS
LIN {X 93.3343,Y 55.1989,Z 108,A 25.6345,B 24.9341,C -1.8755,E1 25.1383,E2 420.0755} C_DIS
LIN {X 94.8947,Y 52.4731,Z 108,A 23.975,B 24.9344,C -1.871,E1 25.1406,E2 421.7371} C_DIS
LIN {X 96.8616,Y 48.7481,Z 108,A 20.9985,B 24.937,C -1.8326,E1 25.1445,E2 424.7883} C_DIS
LIN {X 99.0908,Y 44.0404,Z 108,A 19.0334,B 24.9353,C -1.8585,E1 25.1466,E2 426.6817} C_DIS
Enddeposition()
END
